REGION Network 6: #"PHT Selected"
   RUNG wire#powerrail
      Contact( #DataLogYes )
      I_Contact( #ScadaHmi )
      wire#w1
      I_Contact( #Popup2Enable )
      wire#w2
      I_Contact( #Stop )
      I_Contact( #Fault )
      I_Contact( #ReleaseCheckTime.DONE_BIT )
      wire#w3
      S_Coil( #"PHT Selected" )
   END_RUNG
   RUNG wire#powerrail
      Contact( #StartupMsgYes )
      Contact( #ScadaHmi )
   END_RUNG wire#w1
   RUNG wire#powerrail
      Contact( #Popup2Ack )
      Contact( #Popup2Enable )
   END_RUNG wire#w2
   RUNG wire#powerrail
      Contact( #"PHT Selected" )
      Contact( #Start )
   END_RUNG wire#w2
   RUNG wire#powerrail
      Contact( #Running )
   END_RUNG wire#w2
   RUNG wire#w3
      Coil( #Running )
   END_RUNG
   // the same network as SCL:
   #_w1 := ((((#DataLogYes AND NOT #ScadaHmi) OR (#StartupMsgYes AND #ScadaHmi)) AND NOT #Popup2Enable) OR (#Popup2Ack AND #Popup2Enable) OR (#"PHT Selected" AND #Start) OR #Running) AND NOT #Stop AND NOT #Fault AND NOT #ReleaseCheckTime.DONE_BIT;
   IF #_w1 THEN #"PHT Selected" := TRUE; END_IF;
   #Running := #_w1;
END_REGION

REGION Network 7
   RUNG wire#powerrail
      Contact( #AlwaysTrue )
      wire#w1
      Contact( #"PHT Selected" )
      wire#w2
      R_Coil( #StartLog )
   END_RUNG
   RUNG wire#w1
      I_Contact( #CycleSelected )
   END_RUNG wire#w2
   RUNG wire#w1
      I_Contact( #"PHT Selected" )
      R_Coil( #EndLog )
   END_RUNG
   // the same network as SCL:
   IF #AlwaysTrue AND (#"PHT Selected" OR NOT #CycleSelected) THEN #StartLog := FALSE; END_IF;
   IF #AlwaysTrue AND NOT #"PHT Selected" THEN #EndLog := FALSE; END_IF;
END_REGION

REGION Network 8: OUTPUT ON
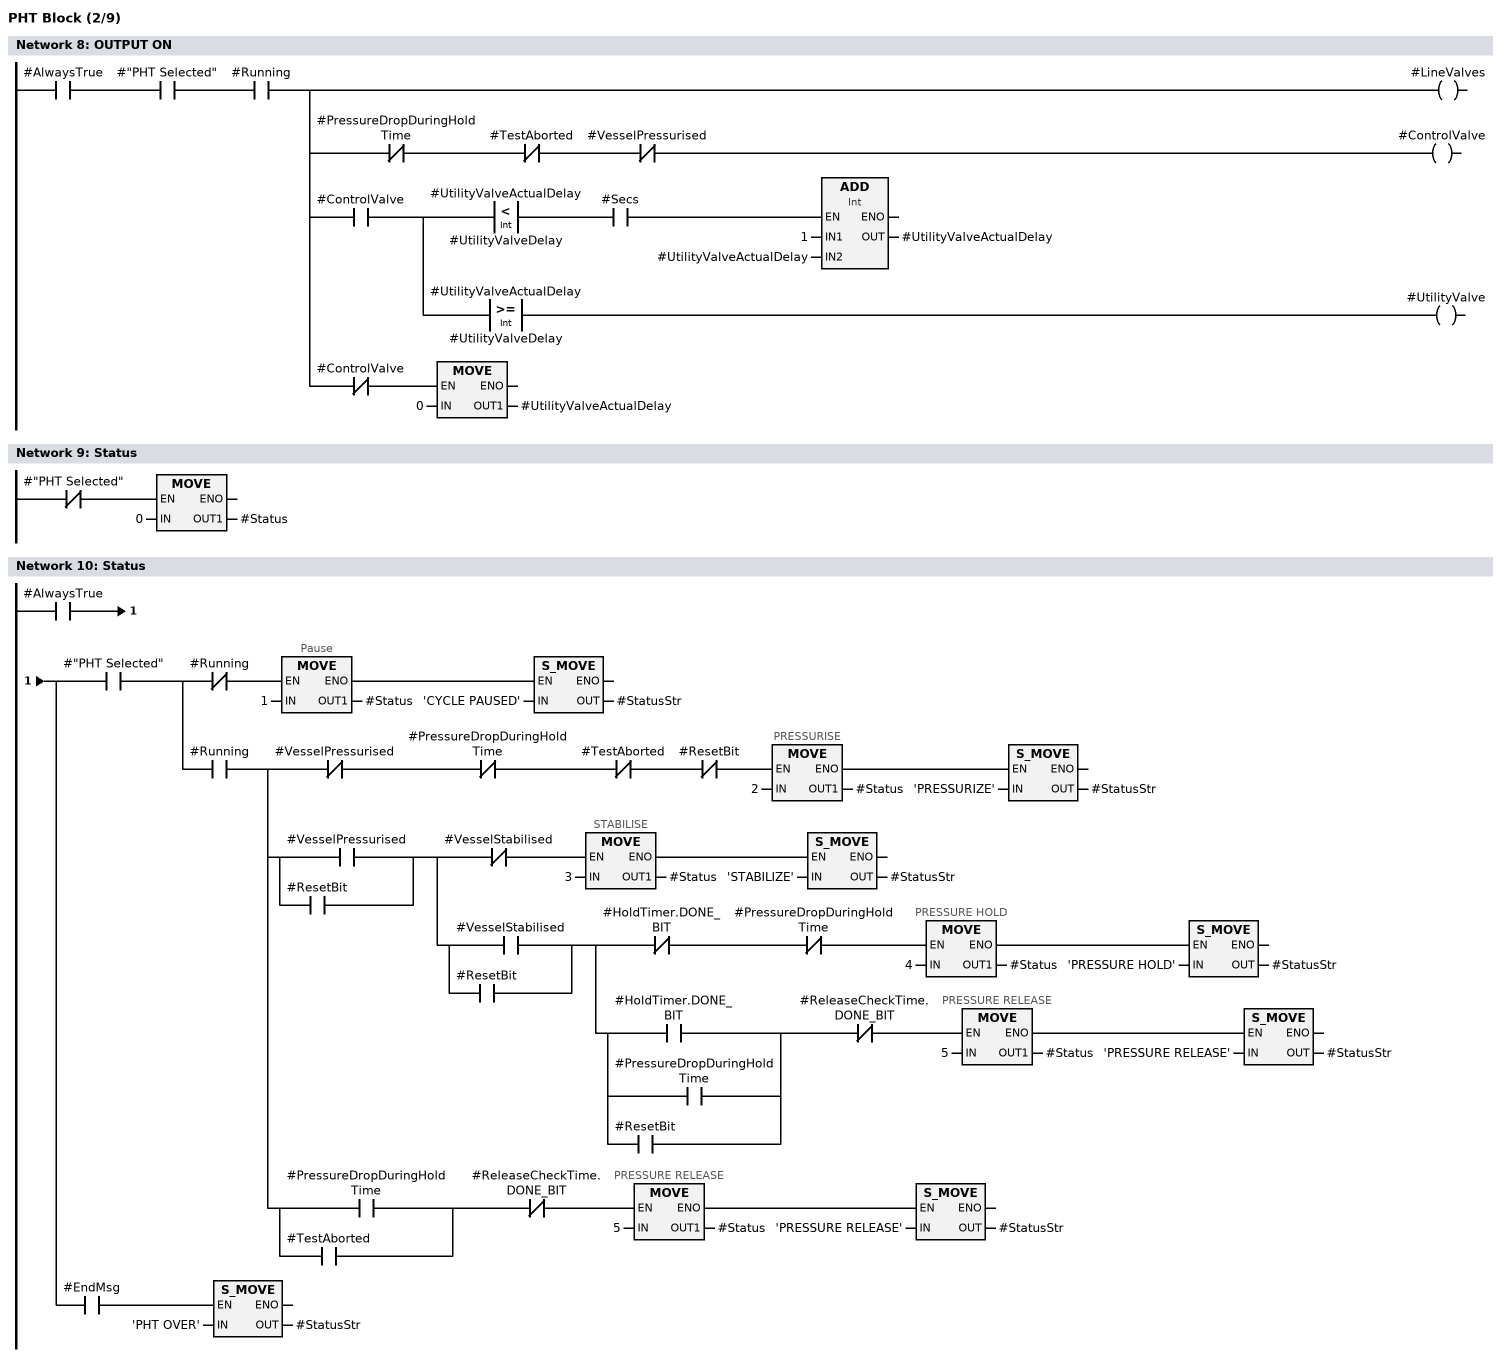
   RUNG wire#powerrail
      Contact( #AlwaysTrue )
      Contact( #"PHT Selected" )
      Contact( #Running )
      wire#w1
      Coil( #LineValves )
   END_RUNG
   RUNG wire#w1
      I_Contact( #PressureDropDuringHoldTime )
      I_Contact( #TestAborted )
      I_Contact( #VesselPressurised )
      Coil( #ControlValve )
   END_RUNG
   RUNG wire#w1
      Contact( #ControlValve )
      wire#w2
      { S7_Templates := "SrcType := Int" } LT_Contact(in1 := #UtilityValveActualDelay, in2 := #UtilityValveDelay)
      Contact( #Secs )
      { S7_Templates := "SrcType := Int" } Add(in1 := 1, in2 := #UtilityValveActualDelay, out => #UtilityValveActualDelay)
   END_RUNG
   RUNG wire#w2
      { S7_Templates := "SrcType := Int" } GE_Contact(in1 := #UtilityValveActualDelay, in2 := #UtilityValveDelay)
      Coil( #UtilityValve )
   END_RUNG
   RUNG wire#w1
      I_Contact( #ControlValve )
      Move(in := 0, out1 => #UtilityValveActualDelay)
   END_RUNG
   // the same network as SCL:
   #LineValves := #AlwaysTrue AND #"PHT Selected" AND #Running;
   #ControlValve := #LineValves AND NOT #PressureDropDuringHoldTime AND NOT #TestAborted AND NOT #VesselPressurised;
   #_w1 := #LineValves AND #ControlValve;
   IF #_w1 AND (#UtilityValveActualDelay < #UtilityValveDelay) AND #Secs THEN
       #UtilityValveActualDelay := 1 + #UtilityValveActualDelay;
   END_IF;
   #UtilityValve := #_w1 AND (#UtilityValveActualDelay >= #UtilityValveDelay);
   IF #LineValves AND NOT #ControlValve THEN #UtilityValveActualDelay := 0; END_IF;
END_REGION

REGION Network 9: Status
   RUNG wire#powerrail
      I_Contact( #"PHT Selected" )
      { S7_GenerateENO := "TRUE" } Move(in := 0, out1 => #Status)
   END_RUNG
   // the same network as SCL:
   IF NOT #"PHT Selected" THEN #Status := 0; END_IF;
END_REGION

REGION Network 10: Status
   RUNG wire#powerrail
      Contact( #AlwaysTrue )
      wire#w1
      Contact( #"PHT Selected" )
      wire#w2
      I_Contact( #Running )
      { S7_GenerateENO := "TRUE" } Move(in := 1, out1 => #Status)   // Pause
      S_Move(in := 'CYCLE PAUSED', out => #StatusStr)
   END_RUNG
   RUNG wire#w2
      Contact( #Running )
      wire#w3
      I_Contact( #VesselPressurised )
      I_Contact( #PressureDropDuringHoldTime )
      I_Contact( #TestAborted )
      I_Contact( #ResetBit )
      { S7_GenerateENO := "TRUE" } Move(in := 2, out1 => #Status)   // PRESSURISE
      S_Move(in := 'PRESSURIZE', out => #StatusStr)
   END_RUNG
   RUNG wire#w3
      Contact( #VesselPressurised )
      wire#w4
      I_Contact( #VesselStabilised )
      { S7_GenerateENO := "TRUE" } Move(in := 3, out1 => #Status)   // STABILISE
      S_Move(in := 'STABILIZE', out => #StatusStr)
   END_RUNG
   RUNG wire#w3
      Contact( #ResetBit )
   END_RUNG wire#w4
   RUNG wire#w4
      Contact( #VesselStabilised )
      wire#w5
      I_Contact( #HoldTimer.DONE_BIT )
      I_Contact( #PressureDropDuringHoldTime )
      { S7_GenerateENO := "TRUE" } Move(in := 4, out1 => #Status)   // PRESSURE HOLD
      S_Move(in := 'PRESSURE HOLD', out => #StatusStr)
   END_RUNG
   RUNG wire#w4
      Contact( #ResetBit )
   END_RUNG wire#w5
   RUNG wire#w5
      Contact( #HoldTimer.DONE_BIT )
      wire#w6
      I_Contact( #ReleaseCheckTime.DONE_BIT )
      { S7_GenerateENO := "TRUE" } Move(in := 5, out1 => #Status)   // PRESSURE RELEASE
      S_Move(in := 'PRESSURE RELEASE', out => #StatusStr)
   END_RUNG
   RUNG wire#w5
      Contact( #PressureDropDuringHoldTime )
   END_RUNG wire#w6
   RUNG wire#w5
      Contact( #ResetBit )
   END_RUNG wire#w6
   RUNG wire#w3
      Contact( #PressureDropDuringHoldTime )
      wire#w7
      I_Contact( #ReleaseCheckTime.DONE_BIT )
      { S7_GenerateENO := "TRUE" } Move(in := 5, out1 => #Status)   // PRESSURE RELEASE
      S_Move(in := 'PRESSURE RELEASE', out => #StatusStr)
   END_RUNG
   RUNG wire#w3
      Contact( #TestAborted )
   END_RUNG wire#w7
   RUNG wire#w1
      Contact( #EndMsg )
      S_Move(in := 'PHT OVER', out => #StatusStr)
   END_RUNG
   // the same network as SCL:
   // ENO of a box is taken as its EN; it also drops when the box reports an error
   #_w1 := #AlwaysTrue AND #"PHT Selected";
   IF #_w1 AND NOT #Running THEN
       #Status := 1;   // Pause
       #StatusStr := 'CYCLE PAUSED';
   END_IF;
   #_w2 := #_w1 AND #Running;
   IF #_w2 AND NOT #VesselPressurised AND NOT #PressureDropDuringHoldTime AND NOT #TestAborted AND NOT #ResetBit THEN
       #Status := 2;   // PRESSURISE
       #StatusStr := 'PRESSURIZE';
   END_IF;
   #_w3 := #_w2 AND (#VesselPressurised OR #ResetBit);
   IF #_w3 AND NOT #VesselStabilised THEN
       #Status := 3;   // STABILISE
       #StatusStr := 'STABILIZE';
   END_IF;
   #_w4 := #_w3 AND (#VesselStabilised OR #ResetBit);
   IF #_w4 AND NOT #HoldTimer.DONE_BIT AND NOT #PressureDropDuringHoldTime THEN
       #Status := 4;   // PRESSURE HOLD
       #StatusStr := 'PRESSURE HOLD';
   END_IF;
   IF #_w4 AND (#HoldTimer.DONE_BIT OR #PressureDropDuringHoldTime OR #ResetBit) AND NOT #ReleaseCheckTime.DONE_BIT THEN
       #Status := 5;   // PRESSURE RELEASE
       #StatusStr := 'PRESSURE RELEASE';
   END_IF;
   IF #_w2 AND (#PressureDropDuringHoldTime OR #TestAborted) AND NOT #ReleaseCheckTime.DONE_BIT THEN
       #Status := 5;   // PRESSURE RELEASE
       #StatusStr := 'PRESSURE RELEASE';
   END_IF;
   IF #AlwaysTrue AND #EndMsg THEN #StatusStr := 'PHT OVER'; END_IF;
END_REGION

REGION Network 11: Delays for opening drain valves
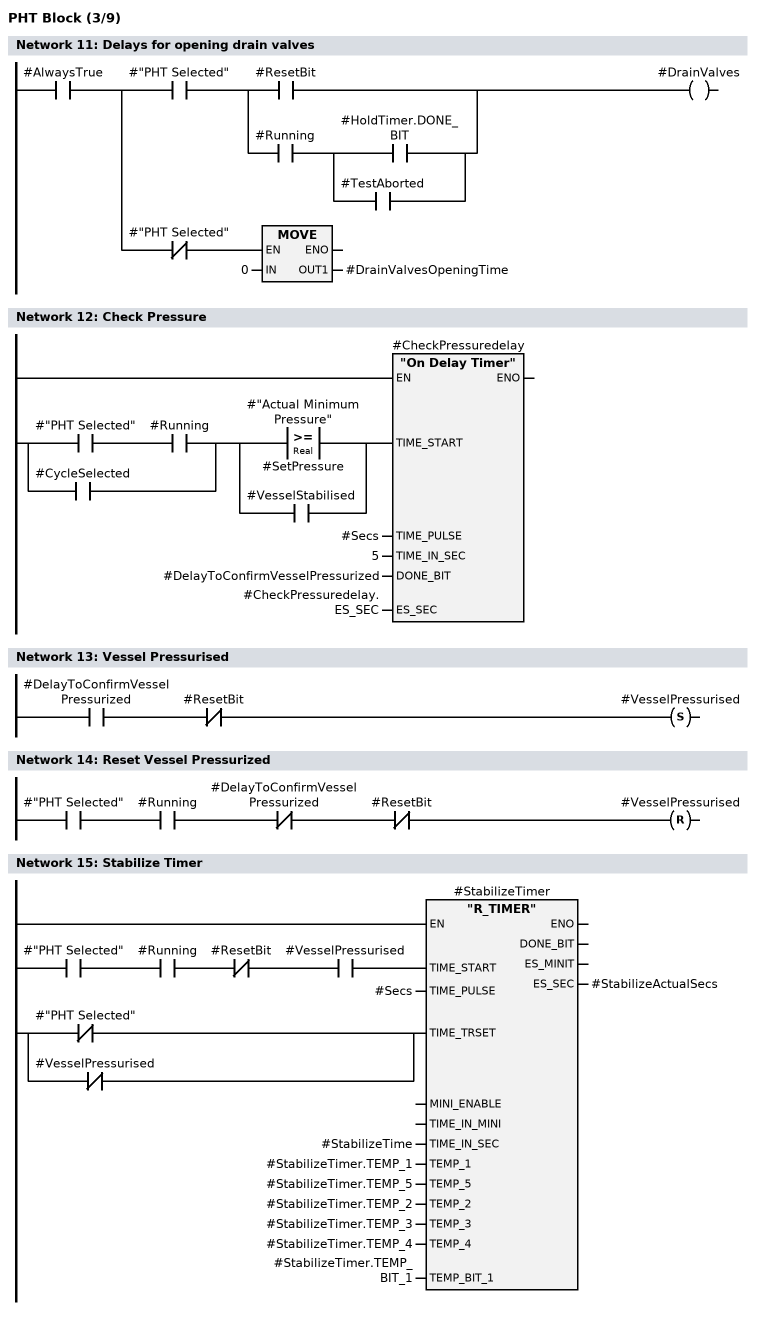
   RUNG wire#powerrail
      Contact( #AlwaysTrue )
      wire#w1
      Contact( #"PHT Selected" )
      wire#w2
      Contact( #ResetBit )
      wire#w3
      Coil( #DrainValves )
   END_RUNG
   RUNG wire#w2
      Contact( #Running )
      wire#w4
      Contact( #HoldTimer.DONE_BIT )
   END_RUNG wire#w3
   RUNG wire#w4
      Contact( #TestAborted )
   END_RUNG wire#w3
   RUNG wire#w1
      I_Contact( #"PHT Selected" )
      { S7_GenerateENO := "TRUE" } Move(in := 0, out1 => #DrainValvesOpeningTime)
   END_RUNG
   // the same network as SCL:
   #DrainValves := #AlwaysTrue AND #"PHT Selected" AND (#ResetBit OR (#Running AND (#HoldTimer.DONE_BIT OR #TestAborted)));
   IF #AlwaysTrue AND NOT #"PHT Selected" THEN #DrainValvesOpeningTime := 0; END_IF;
END_REGION

REGION Network 12: Check Pressure
   RUNG wire#powerrail
      #CheckPressuredelay(TIME_START := wire#w2, TIME_PULSE := #Secs, TIME_IN_SEC := 5, DONE_BIT := #DelayToConfirmVesselPressurized, ES_SEC := #CheckPressuredelay.ES_SEC)
   END_RUNG
   RUNG wire#powerrail
      Contact( #"PHT Selected" )
      Contact( #Running )
      wire#w1
      { S7_Templates := "SrcType := Real" } GE_Contact(in1 := #"Actual Minimum Pressure", in2 := #SetPressure)
   END_RUNG wire#w2
   RUNG wire#powerrail
      Contact( #CycleSelected )
   END_RUNG wire#w1
   RUNG wire#w1
      Contact( #VesselStabilised )
   END_RUNG wire#w2
   // the same network as SCL:
   #CheckPressuredelay(TIME_START := ((#"PHT Selected" AND #Running) OR #CycleSelected) AND ((#"Actual Minimum Pressure" >= #SetPressure) OR #VesselStabilised),   // "On Delay Timer"
                       TIME_PULSE := #Secs,
                       TIME_IN_SEC := 5,
                       DONE_BIT := #DelayToConfirmVesselPressurized,
                       ES_SEC := #CheckPressuredelay.ES_SEC);
END_REGION

REGION Network 13: Vessel Pressurised
   RUNG wire#powerrail
      Contact( #DelayToConfirmVesselPressurized )
      I_Contact( #ResetBit )
      S_Coil( #VesselPressurised )
   END_RUNG
   // the same network as SCL:
   IF #DelayToConfirmVesselPressurized AND NOT #ResetBit THEN #VesselPressurised := TRUE; END_IF;
END_REGION

REGION Network 14: Reset Vessel Pressurized
   RUNG wire#powerrail
      Contact( #"PHT Selected" )
      Contact( #Running )
      I_Contact( #DelayToConfirmVesselPressurized )
      I_Contact( #ResetBit )
      R_Coil( #VesselPressurised )
   END_RUNG
   // the same network as SCL:
   IF #"PHT Selected" AND #Running AND NOT #DelayToConfirmVesselPressurized AND NOT #ResetBit THEN
       #VesselPressurised := FALSE;
   END_IF;
END_REGION

REGION Network 15: Stabilize Timer
   RUNG wire#powerrail
      #StabilizeTimer(TIME_START := wire#w1, TIME_TRSET := wire#w2, TIME_PULSE := #Secs, MINI_ENABLE :=, TIME_IN_MINI :=, TIME_IN_SEC := #StabilizeTime, TEMP_1 := #StabilizeTimer.TEMP_1, TEMP_5 := #StabilizeTimer.TEMP_5, TEMP_2 := #StabilizeTimer.TEMP_2, TEMP_3 := #StabilizeTimer.TEMP_3, TEMP_4 := #StabilizeTimer.TEMP_4, TEMP_BIT_1 := #StabilizeTimer.TEMP_BIT_1, DONE_BIT =>, ES_MINIT =>, ES_SEC => #StabilizeActualSecs)
   END_RUNG
   RUNG wire#powerrail
      Contact( #"PHT Selected" )
      Contact( #Running )
      I_Contact( #ResetBit )
      Contact( #VesselPressurised )
   END_RUNG wire#w1
   RUNG wire#powerrail
      I_Contact( #"PHT Selected" )
   END_RUNG wire#w2
   RUNG wire#powerrail
      I_Contact( #VesselPressurised )
   END_RUNG wire#w2
   // the same network as SCL:
   #StabilizeTimer(TIME_START := #"PHT Selected" AND #Running AND NOT #ResetBit AND #VesselPressurised,   // "R_TIMER"
                   TIME_PULSE := #Secs,
                   TIME_TRSET := NOT #"PHT Selected" OR NOT #VesselPressurised,
                   TIME_IN_SEC := #StabilizeTime,
                   TEMP_1 := #StabilizeTimer.TEMP_1,
                   TEMP_5 := #StabilizeTimer.TEMP_5,
                   TEMP_2 := #StabilizeTimer.TEMP_2,
                   TEMP_3 := #StabilizeTimer.TEMP_3,
                   TEMP_4 := #StabilizeTimer.TEMP_4,
                   TEMP_BIT_1 := #StabilizeTimer.TEMP_BIT_1,
                   ES_SEC => #StabilizeActualSecs);
END_REGION

REGION Network 16: Check Pressure During Stabilize
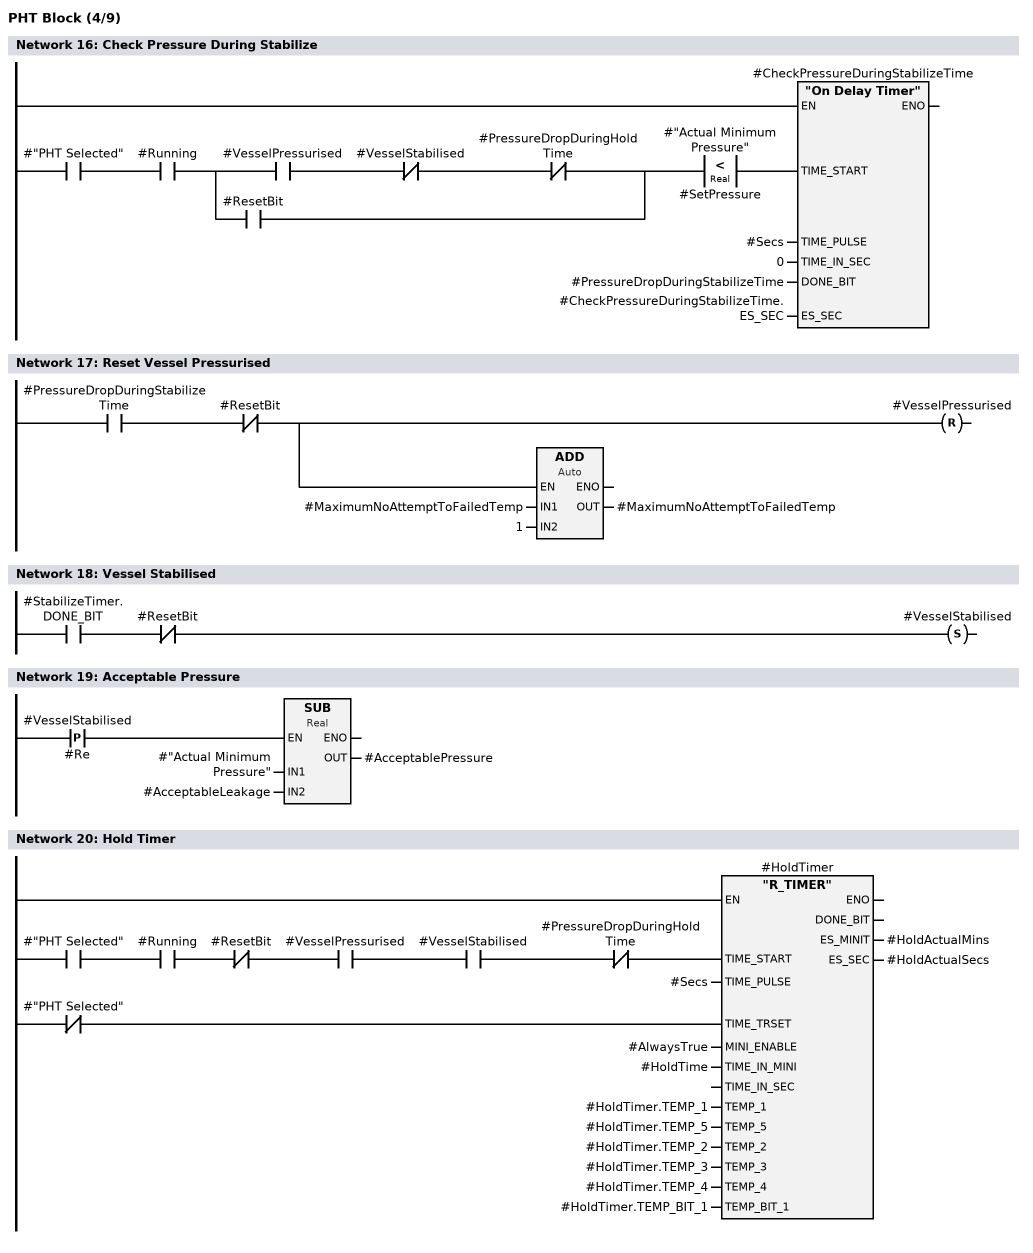
   RUNG wire#powerrail
      #CheckPressureDuringStabilizeTime(TIME_START := wire#w3, TIME_PULSE := #Secs, TIME_IN_SEC := 0, DONE_BIT := #PressureDropDuringStabilizeTime, ES_SEC := #CheckPressureDuringStabilizeTime.ES_SEC)
   END_RUNG
   RUNG wire#powerrail
      Contact( #"PHT Selected" )
      Contact( #Running )
      wire#w1
      Contact( #VesselPressurised )
      I_Contact( #VesselStabilised )
      I_Contact( #PressureDropDuringHoldTime )
      wire#w2
      { S7_Templates := "SrcType := Real" } LT_Contact(in1 := #"Actual Minimum Pressure", in2 := #SetPressure)
   END_RUNG wire#w3
   RUNG wire#w1
      Contact( #ResetBit )
   END_RUNG wire#w2
   // the same network as SCL:
   #CheckPressureDuringStabilizeTime(TIME_START := #"PHT Selected" AND #Running AND ((#VesselPressurised AND NOT #VesselStabilised AND NOT #PressureDropDuringHoldTime) OR #ResetBit) AND (#"Actual Minimum Pressure" < #SetPressure),   // "On Delay Timer"
                           TIME_PULSE := #Secs,
                           TIME_IN_SEC := 0,
                           DONE_BIT := #PressureDropDuringStabilizeTime,
                           ES_SEC := #CheckPressureDuringStabilizeTime.ES_SEC);
END_REGION

REGION Network 17: Reset Vessel Pressurised
   RUNG wire#powerrail
      Contact( #PressureDropDuringStabilizeTime )
      I_Contact( #ResetBit )
      wire#w1
      R_Coil( #VesselPressurised )
   END_RUNG
   RUNG wire#w1
      Add(in1 := #MaximumNoAttemptToFailedTemp, in2 := 1, out => #MaximumNoAttemptToFailedTemp)
   END_RUNG
   // the same network as SCL:
   IF #PressureDropDuringStabilizeTime AND NOT #ResetBit THEN
       #VesselPressurised := FALSE;
       #MaximumNoAttemptToFailedTemp := #MaximumNoAttemptToFailedTemp + 1;
   END_IF;
END_REGION

REGION Network 18: Vessel Stabilised
   RUNG wire#powerrail
      Contact( #StabilizeTimer.DONE_BIT )
      I_Contact( #ResetBit )
      S_Coil( #VesselStabilised )
   END_RUNG
   // the same network as SCL:
   IF #StabilizeTimer.DONE_BIT AND NOT #ResetBit THEN #VesselStabilised := TRUE; END_IF;
END_REGION

REGION Network 19: Acceptable Pressure
   RUNG wire#powerrail
      P_Contact(operand := #VesselStabilised, bit := #Re)
      { S7_Templates := "SrcType := Real"; S7_GenerateENO := "TRUE" } Sub(in1 := #"Actual Minimum Pressure", in2 := #AcceptableLeakage, out => #AcceptablePressure)
   END_RUNG
   // the same network as SCL:
   #_w1 := #VesselStabilised AND NOT #Re;   // rising edge of #VesselStabilised
   #Re := #VesselStabilised;
   IF #_w1 THEN #AcceptablePressure := #"Actual Minimum Pressure" - #AcceptableLeakage; END_IF;
END_REGION

REGION Network 20: Hold Timer
   RUNG wire#powerrail
      #HoldTimer(TIME_START := wire#w1, TIME_TRSET := wire#w2, TIME_PULSE := #Secs, MINI_ENABLE := #AlwaysTrue, TIME_IN_MINI := #HoldTime, TIME_IN_SEC :=, TEMP_1 := #HoldTimer.TEMP_1, TEMP_5 := #HoldTimer.TEMP_5, TEMP_2 := #HoldTimer.TEMP_2, TEMP_3 := #HoldTimer.TEMP_3, TEMP_4 := #HoldTimer.TEMP_4, TEMP_BIT_1 := #HoldTimer.TEMP_BIT_1, DONE_BIT =>, ES_MINIT => #HoldActualMins, ES_SEC => #HoldActualSecs)
   END_RUNG
   RUNG wire#powerrail
      Contact( #"PHT Selected" )
      Contact( #Running )
      I_Contact( #ResetBit )
      Contact( #VesselPressurised )
      Contact( #VesselStabilised )
      I_Contact( #PressureDropDuringHoldTime )
   END_RUNG wire#w1
   RUNG wire#powerrail
      I_Contact( #"PHT Selected" )
   END_RUNG wire#w2
   // the same network as SCL:
   #HoldTimer(TIME_START := #"PHT Selected" AND #Running AND NOT #ResetBit AND #VesselPressurised AND #VesselStabilised AND NOT #PressureDropDuringHoldTime,   // "R_TIMER"
              TIME_PULSE := #Secs,
              TIME_TRSET := NOT #"PHT Selected",
              MINI_ENABLE := #AlwaysTrue,
              TIME_IN_MINI := #HoldTime,
              TEMP_1 := #HoldTimer.TEMP_1,
              TEMP_5 := #HoldTimer.TEMP_5,
              TEMP_2 := #HoldTimer.TEMP_2,
              TEMP_3 := #HoldTimer.TEMP_3,
              TEMP_4 := #HoldTimer.TEMP_4,
              TEMP_BIT_1 := #HoldTimer.TEMP_BIT_1,
              ES_MINIT => #HoldActualMins,
              ES_SEC => #HoldActualSecs);
END_REGION

REGION Network 21: Check Pressure to abort Cycle during Hold Time
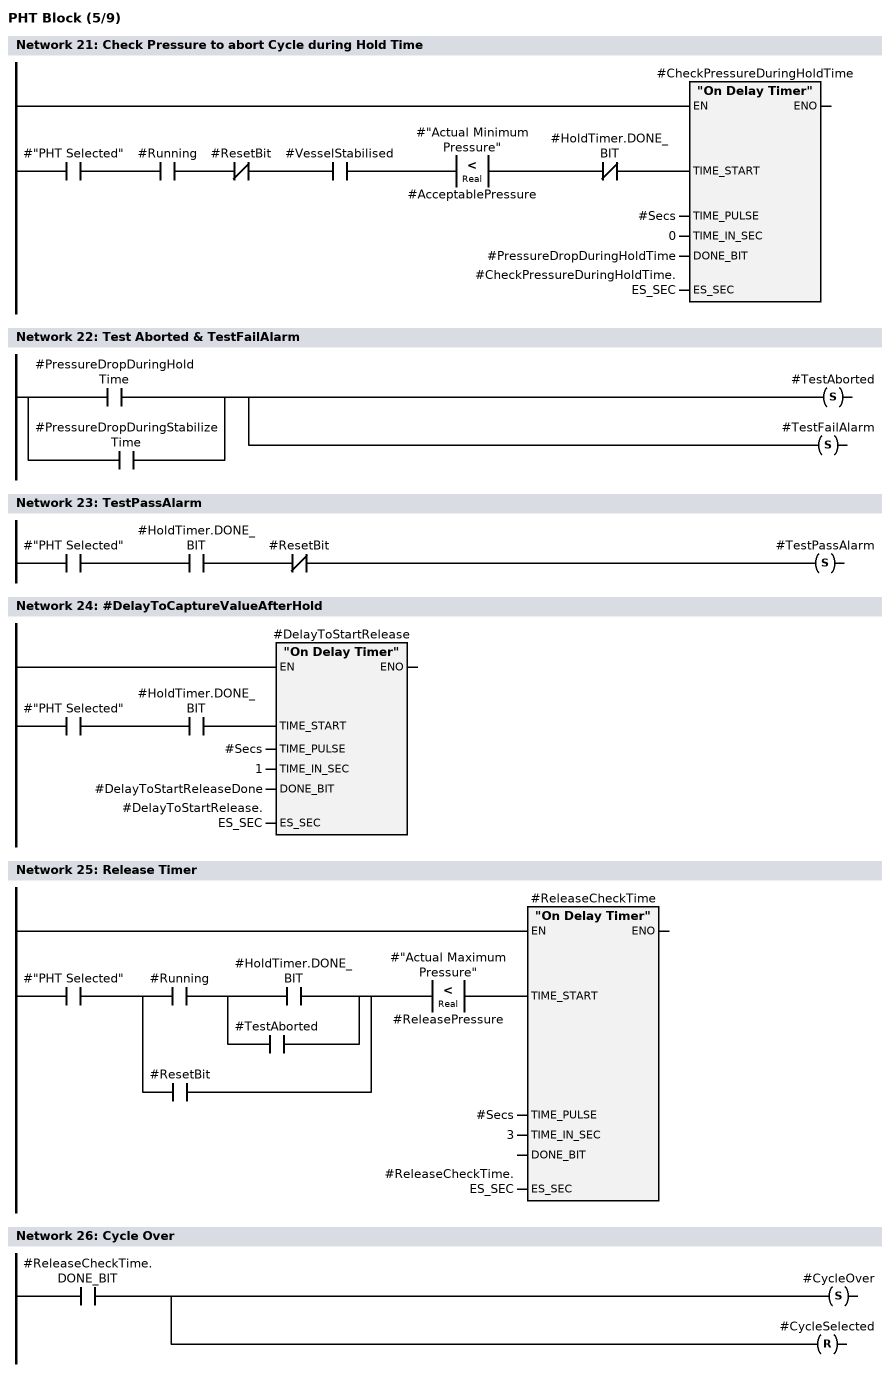
   RUNG wire#powerrail
      #CheckPressureDuringHoldTime(TIME_START := wire#w1, TIME_PULSE := #Secs, TIME_IN_SEC := 0, DONE_BIT := #PressureDropDuringHoldTime, ES_SEC := #CheckPressureDuringHoldTime.ES_SEC)
   END_RUNG
   RUNG wire#powerrail
      Contact( #"PHT Selected" )
      Contact( #Running )
      I_Contact( #ResetBit )
      Contact( #VesselStabilised )
      { S7_Templates := "SrcType := Real" } LT_Contact(in1 := #"Actual Minimum Pressure", in2 := #AcceptablePressure)
      I_Contact( #HoldTimer.DONE_BIT )
   END_RUNG wire#w1
   // the same network as SCL:
   #CheckPressureDuringHoldTime(TIME_START := #"PHT Selected" AND #Running AND NOT #ResetBit AND #VesselStabilised AND (#"Actual Minimum Pressure" < #AcceptablePressure) AND NOT #HoldTimer.DONE_BIT,   // "On Delay Timer"
                           TIME_PULSE := #Secs,
                           TIME_IN_SEC := 0,
                           DONE_BIT := #PressureDropDuringHoldTime,
                           ES_SEC := #CheckPressureDuringHoldTime.ES_SEC);
END_REGION

REGION Network 22: Test Aborted & TestFailAlarm
   RUNG wire#powerrail
      Contact( #PressureDropDuringHoldTime )
      wire#w1
      S_Coil( #TestAborted )
   END_RUNG
   RUNG wire#powerrail
      Contact( #PressureDropDuringStabilizeTime )
   END_RUNG wire#w1
   RUNG wire#w1
      S_Coil( #TestFailAlarm )
   END_RUNG
   // the same network as SCL:
   IF #PressureDropDuringHoldTime OR #PressureDropDuringStabilizeTime THEN
       #TestAborted := TRUE;
       #TestFailAlarm := TRUE;
   END_IF;
END_REGION

REGION Network 23: TestPassAlarm
   RUNG wire#powerrail
      Contact( #"PHT Selected" )
      Contact( #HoldTimer.DONE_BIT )
      I_Contact( #ResetBit )
      S_Coil( #TestPassAlarm )
   END_RUNG
   // the same network as SCL:
   IF #"PHT Selected" AND #HoldTimer.DONE_BIT AND NOT #ResetBit THEN #TestPassAlarm := TRUE; END_IF;
END_REGION

REGION Network 24: #DelayToCaptureValueAfterHold
   RUNG wire#powerrail
      #DelayToStartRelease(TIME_START := wire#w1, TIME_PULSE := #Secs, TIME_IN_SEC := 1, DONE_BIT := #DelayToStartReleaseDone, ES_SEC := #DelayToStartRelease.ES_SEC)
   END_RUNG
   RUNG wire#powerrail
      Contact( #"PHT Selected" )
      Contact( #HoldTimer.DONE_BIT )
   END_RUNG wire#w1
   // the same network as SCL:
   #DelayToStartRelease(TIME_START := #"PHT Selected" AND #HoldTimer.DONE_BIT,   // "On Delay Timer"
                        TIME_PULSE := #Secs,
                        TIME_IN_SEC := 1,
                        DONE_BIT := #DelayToStartReleaseDone,
                        ES_SEC := #DelayToStartRelease.ES_SEC);
END_REGION

REGION Network 25: Release Timer
   RUNG wire#powerrail
      #ReleaseCheckTime(TIME_START := wire#w4, TIME_PULSE := #Secs, TIME_IN_SEC := 3, DONE_BIT :=, ES_SEC := #ReleaseCheckTime.ES_SEC)
   END_RUNG
   RUNG wire#powerrail
      Contact( #"PHT Selected" )
      wire#w1
      Contact( #Running )
      wire#w2
      Contact( #HoldTimer.DONE_BIT )
      wire#w3
      { S7_Templates := "SrcType := Real" } LT_Contact(in1 := #"Actual Maximum Pressure", in2 := #ReleasePressure)
   END_RUNG wire#w4
   RUNG wire#w2
      Contact( #TestAborted )
   END_RUNG wire#w3
   RUNG wire#w1
      Contact( #ResetBit )
   END_RUNG wire#w3
   // the same network as SCL:
   #ReleaseCheckTime(TIME_START := #"PHT Selected" AND ((#Running AND (#HoldTimer.DONE_BIT OR #TestAborted)) OR #ResetBit) AND (#"Actual Maximum Pressure" < #ReleasePressure),   // "On Delay Timer"
                     TIME_PULSE := #Secs,
                     TIME_IN_SEC := 3,
                     ES_SEC := #ReleaseCheckTime.ES_SEC);
END_REGION

REGION Network 26: Cycle Over
   RUNG wire#powerrail
      Contact( #ReleaseCheckTime.DONE_BIT )
      wire#w1
      S_Coil( #CycleOver )
   END_RUNG
   RUNG wire#w1
      R_Coil( #CycleSelected )
   END_RUNG
   // the same network as SCL:
   IF #ReleaseCheckTime.DONE_BIT THEN
       #CycleOver := TRUE;
       #CycleSelected := FALSE;
   END_IF;
END_REGION

REGION Network 27: Alarm Ack
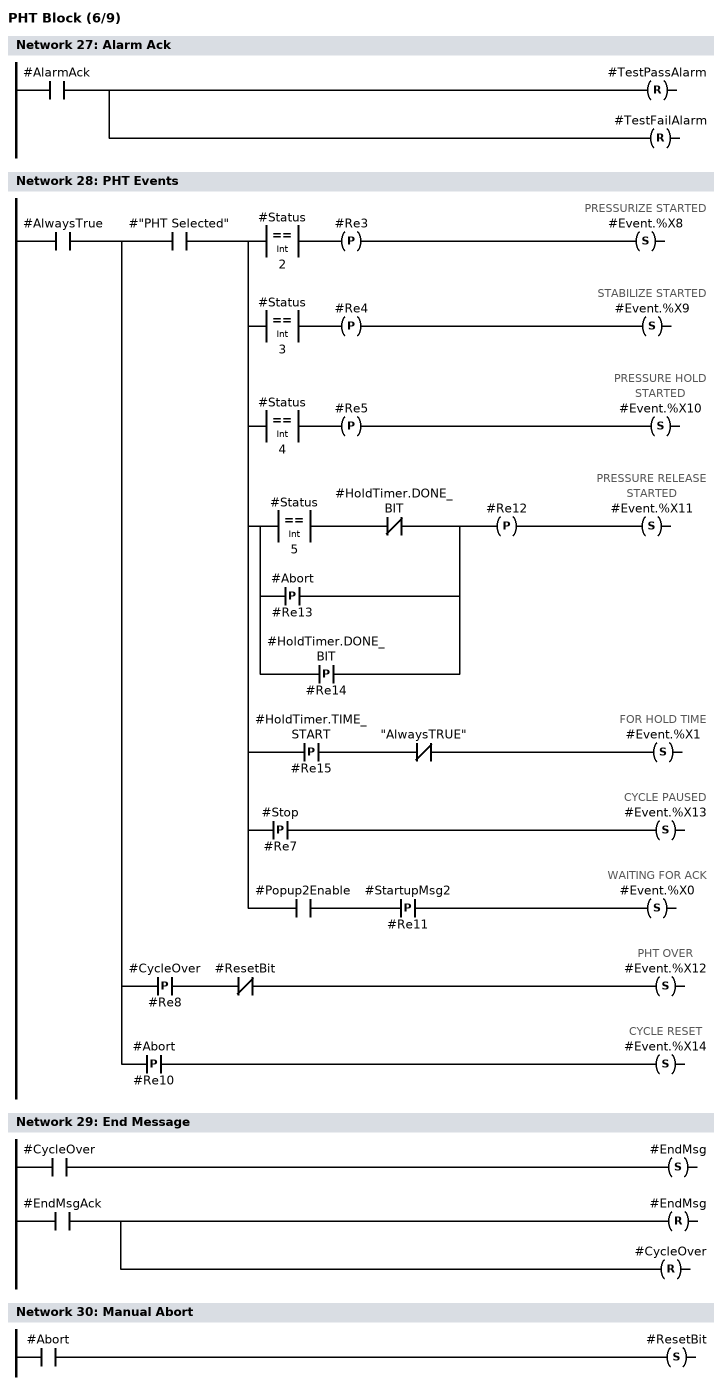
   RUNG wire#powerrail
      Contact( #AlarmAck )
      wire#w1
      R_Coil( #TestPassAlarm )
   END_RUNG
   RUNG wire#w1
      R_Coil( #TestFailAlarm )
   END_RUNG
   // the same network as SCL:
   IF #AlarmAck THEN
       #TestPassAlarm := FALSE;
       #TestFailAlarm := FALSE;
   END_IF;
END_REGION

REGION Network 28: PHT Events
   RUNG wire#powerrail
      Contact( #AlwaysTrue )
      wire#w1
      Contact( #"PHT Selected" )
      wire#w2
      { S7_Templates := "SrcType := Int" } EQ_Contact(in1 := #Status, in2 := 2)
      P_Trig( #Re3 )
      S_Coil( #Event.%X8 )   // PRESSURIZE STARTED
   END_RUNG
   RUNG wire#w2
      { S7_Templates := "SrcType := Int" } EQ_Contact(in1 := #Status, in2 := 3)
      P_Trig( #Re4 )
      S_Coil( #Event.%X9 )   // STABILIZE STARTED
   END_RUNG
   RUNG wire#w2
      { S7_Templates := "SrcType := Int" } EQ_Contact(in1 := #Status, in2 := 4)
      P_Trig( #Re5 )
      S_Coil( #Event.%X10 )   // PRESSURE HOLD STARTED
   END_RUNG
   RUNG wire#w2
      { S7_Templates := "SrcType := Int" } EQ_Contact(in1 := #Status, in2 := 5)
      I_Contact( #HoldTimer.DONE_BIT )
      wire#w3
      P_Trig( #Re12 )
      S_Coil( #Event.%X11 )   // PRESSURE RELEASE STARTED
   END_RUNG
   RUNG wire#w2
      P_Contact(operand := #Abort, bit := #Re13)
   END_RUNG wire#w3
   RUNG wire#w2
      P_Contact(operand := #HoldTimer.DONE_BIT, bit := #Re14)
   END_RUNG wire#w3
   RUNG wire#w2
      P_Contact(operand := #HoldTimer.TIME_START, bit := #Re15)
      I_Contact( "AlwaysTRUE" )
      S_Coil( #Event.%X1 )   // FOR HOLD TIME
   END_RUNG
   RUNG wire#w2
      P_Contact(operand := #Stop, bit := #Re7)
      S_Coil( #Event.%X13 )   // CYCLE PAUSED
   END_RUNG
   RUNG wire#w2
      Contact( #Popup2Enable )
      P_Contact(operand := #StartupMsg2, bit := #Re11)
      S_Coil( #Event.%X0 )   // WAITING FOR ACK
   END_RUNG
   RUNG wire#w1
      P_Contact(operand := #CycleOver, bit := #Re8)
      I_Contact( #ResetBit )
      S_Coil( #Event.%X12 )   // PHT OVER
   END_RUNG
   RUNG wire#w1
      P_Contact(operand := #Abort, bit := #Re10)
      S_Coil( #Event.%X14 )   // CYCLE RESET
   END_RUNG
   // the same network as SCL:
   #_w1 := #AlwaysTrue AND #"PHT Selected";
   #_w2 := #_w1 AND (#Status = 2);
   #_w3 := #_w2 AND NOT #Re3;   // rising edge
   #Re3 := #_w2;
   IF #_w3 THEN
       #Event.%X8 := TRUE;   // PRESSURIZE STARTED
   END_IF;
   #_w4 := #_w1 AND (#Status = 3);
   #_w5 := #_w4 AND NOT #Re4;   // rising edge
   #Re4 := #_w4;
   IF #_w5 THEN
       #Event.%X9 := TRUE;   // STABILIZE STARTED
   END_IF;
   #_w6 := #_w1 AND (#Status = 4);
   #_w7 := #_w6 AND NOT #Re5;   // rising edge
   #Re5 := #_w6;
   IF #_w7 THEN
       #Event.%X10 := TRUE;   // PRESSURE HOLD STARTED
   END_IF;
   #_w8 := #_w1 AND #Abort AND NOT #Re13;   // rising edge of #Abort
   #Re13 := #Abort;
   #_w9 := #_w1 AND #HoldTimer.DONE_BIT AND NOT #Re14;   // rising edge of #HoldTimer.DONE_BIT
   #Re14 := #HoldTimer.DONE_BIT;
   #_w10 := (#_w1 AND (#Status = 5) AND NOT #HoldTimer.DONE_BIT) OR #_w8 OR #_w9;
   #_w11 := #_w10 AND NOT #Re12;   // rising edge
   #Re12 := #_w10;
   IF #_w11 THEN
       #Event.%X11 := TRUE;   // PRESSURE RELEASE STARTED
   END_IF;
   #_w12 := #_w1 AND #HoldTimer.TIME_START AND NOT #Re15;   // rising edge of #HoldTimer.TIME_START
   #Re15 := #HoldTimer.TIME_START;
   IF #_w12 AND NOT "AlwaysTRUE" THEN
       #Event.%X1 := TRUE;   // FOR HOLD TIME
   END_IF;
   #_w13 := #_w1 AND #Stop AND NOT #Re7;   // rising edge of #Stop
   #Re7 := #Stop;
   IF #_w13 THEN
       #Event.%X13 := TRUE;   // CYCLE PAUSED
   END_IF;
   #_w14 := #_w1 AND #Popup2Enable AND #StartupMsg2 AND NOT #Re11;   // rising edge of #StartupMsg2
   #Re11 := #StartupMsg2;
   IF #_w14 THEN
       #Event.%X0 := TRUE;   // WAITING FOR ACK
   END_IF;
   #_w15 := #AlwaysTrue AND #CycleOver AND NOT #Re8;   // rising edge of #CycleOver
   #Re8 := #CycleOver;
   IF #_w15 AND NOT #ResetBit THEN
       #Event.%X12 := TRUE;   // PHT OVER
   END_IF;
   #_w16 := #AlwaysTrue AND #Abort AND NOT #Re10;   // rising edge of #Abort
   #Re10 := #Abort;
   IF #_w16 THEN
       #Event.%X14 := TRUE;   // CYCLE RESET
   END_IF;
END_REGION

REGION Network 29: End Message
   RUNG wire#powerrail
      Contact( #CycleOver )
      S_Coil( #EndMsg )
   END_RUNG
   RUNG wire#powerrail
      Contact( #EndMsgAck )
      wire#w1
      R_Coil( #EndMsg )
   END_RUNG
   RUNG wire#w1
      R_Coil( #CycleOver )
   END_RUNG
   // the same network as SCL:
   IF #CycleOver THEN #EndMsg := TRUE; END_IF;
   IF #EndMsgAck THEN
       #EndMsg := FALSE;
       #CycleOver := FALSE;
   END_IF;
END_REGION

REGION Network 30: Manual Abort
   RUNG wire#powerrail
      Contact( #Abort )
      S_Coil( #ResetBit )
   END_RUNG
   // the same network as SCL:
   IF #Abort THEN #ResetBit := TRUE; END_IF;
END_REGION

REGION Network 31: Reset
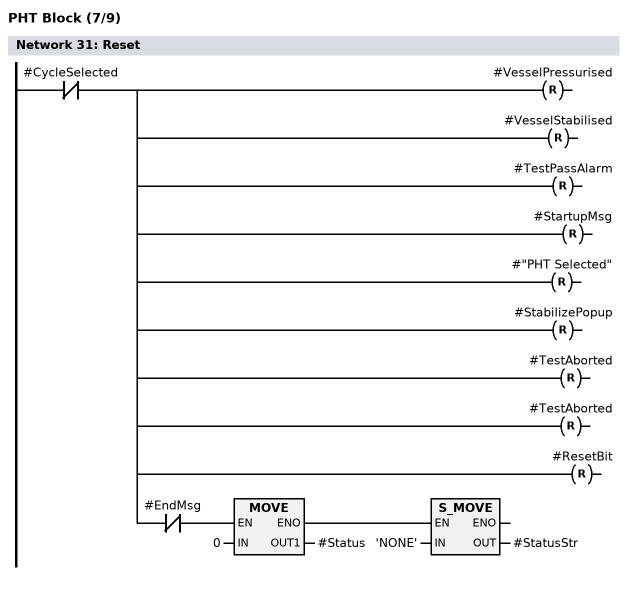
   RUNG wire#powerrail
      I_Contact( #CycleSelected )
      wire#w1
      R_Coil( #VesselPressurised )
   END_RUNG
   RUNG wire#w1
      R_Coil( #VesselStabilised )
   END_RUNG
   RUNG wire#w1
      R_Coil( #TestPassAlarm )
   END_RUNG
   RUNG wire#w1
      R_Coil( #StartupMsg )
   END_RUNG
   RUNG wire#w1
      R_Coil( #"PHT Selected" )
   END_RUNG
   RUNG wire#w1
      R_Coil( #StabilizePopup )
   END_RUNG
   RUNG wire#w1
      R_Coil( #TestAborted )
   END_RUNG
   RUNG wire#w1
      R_Coil( #TestAborted )
   END_RUNG
   RUNG wire#w1
      R_Coil( #ResetBit )
   END_RUNG
   RUNG wire#w1
      I_Contact( #EndMsg )
      { S7_GenerateENO := "TRUE" } Move(in := 0, out1 => #Status)
      S_Move(in := 'NONE', out => #StatusStr)
   END_RUNG
   // the same network as SCL:
   // ENO of a box is taken as its EN; it also drops when the box reports an error
   IF NOT #CycleSelected THEN
       #VesselPressurised := FALSE;
       #VesselStabilised := FALSE;
       #TestPassAlarm := FALSE;
       #StartupMsg := FALSE;
       #"PHT Selected" := FALSE;
       #StabilizePopup := FALSE;
       #TestAborted := FALSE;
       #TestAborted := FALSE;
       #ResetBit := FALSE;
   END_IF;
   IF NOT #CycleSelected AND NOT #EndMsg THEN
       #Status := 0;
       #StatusStr := 'NONE';
   END_IF;
END_REGION

REGION Network 32: Event reset
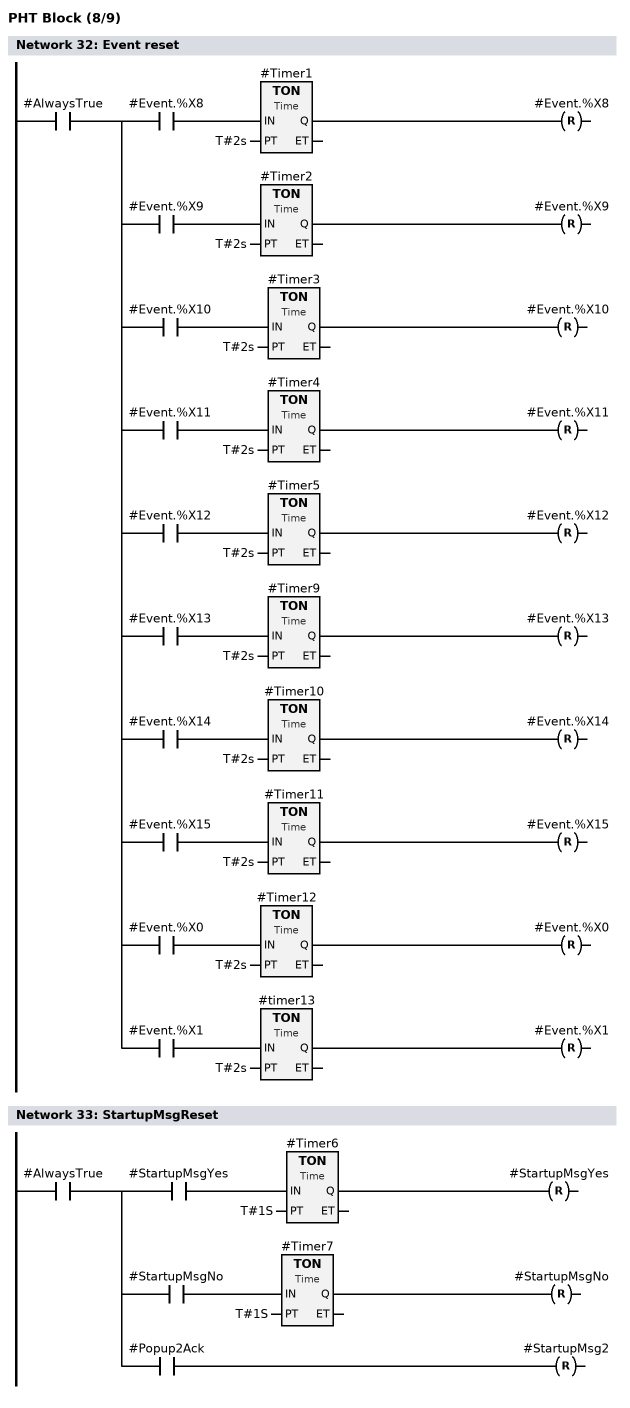
   RUNG wire#powerrail
      Contact( #AlwaysTrue )
      wire#w1
      Contact( #Event.%X8 )
      { S7_Templates := "time_type := Time" } #Timer1.TON(pt := T#2s, et =>)
      R_Coil( #Event.%X8 )
   END_RUNG
   RUNG wire#w1
      Contact( #Event.%X9 )
      { S7_Templates := "time_type := Time" } #Timer2.TON(pt := T#2s, et =>)
      R_Coil( #Event.%X9 )
   END_RUNG
   RUNG wire#w1
      Contact( #Event.%X10 )
      { S7_Templates := "time_type := Time" } #Timer3.TON(pt := T#2s, et =>)
      R_Coil( #Event.%X10 )
   END_RUNG
   RUNG wire#w1
      Contact( #Event.%X11 )
      { S7_Templates := "time_type := Time" } #Timer4.TON(pt := T#2s, et =>)
      R_Coil( #Event.%X11 )
   END_RUNG
   RUNG wire#w1
      Contact( #Event.%X12 )
      { S7_Templates := "time_type := Time" } #Timer5.TON(pt := T#2s, et =>)
      R_Coil( #Event.%X12 )
   END_RUNG
   RUNG wire#w1
      Contact( #Event.%X13 )
      { S7_Templates := "time_type := Time" } #Timer9.TON(pt := T#2s, et =>)
      R_Coil( #Event.%X13 )
   END_RUNG
   RUNG wire#w1
      Contact( #Event.%X14 )
      { S7_Templates := "time_type := Time" } #Timer10.TON(pt := T#2s, et =>)
      R_Coil( #Event.%X14 )
   END_RUNG
   RUNG wire#w1
      Contact( #Event.%X15 )
      { S7_Templates := "time_type := Time" } #Timer11.TON(pt := T#2s, et =>)
      R_Coil( #Event.%X15 )
   END_RUNG
   RUNG wire#w1
      Contact( #Event.%X0 )
      { S7_Templates := "time_type := Time" } #Timer12.TON(pt := T#2s, et =>)
      R_Coil( #Event.%X0 )
   END_RUNG
   RUNG wire#w1
      Contact( #Event.%X1 )
      { S7_Templates := "time_type := Time" } #timer13.TON(pt := T#2s, et =>)
      R_Coil( #Event.%X1 )
   END_RUNG
   // the same network as SCL:
   #Timer1(IN := #AlwaysTrue AND #Event.%X8, PT := T#2s);   // TON
   IF #Timer1.Q THEN #Event.%X8 := FALSE; END_IF;
   #Timer2(IN := #AlwaysTrue AND #Event.%X9, PT := T#2s);   // TON
   IF #Timer2.Q THEN #Event.%X9 := FALSE; END_IF;
   #Timer3(IN := #AlwaysTrue AND #Event.%X10, PT := T#2s);   // TON
   IF #Timer3.Q THEN #Event.%X10 := FALSE; END_IF;
   #Timer4(IN := #AlwaysTrue AND #Event.%X11, PT := T#2s);   // TON
   IF #Timer4.Q THEN #Event.%X11 := FALSE; END_IF;
   #Timer5(IN := #AlwaysTrue AND #Event.%X12, PT := T#2s);   // TON
   IF #Timer5.Q THEN #Event.%X12 := FALSE; END_IF;
   #Timer9(IN := #AlwaysTrue AND #Event.%X13, PT := T#2s);   // TON
   IF #Timer9.Q THEN #Event.%X13 := FALSE; END_IF;
   #Timer10(IN := #AlwaysTrue AND #Event.%X14, PT := T#2s);   // TON
   IF #Timer10.Q THEN #Event.%X14 := FALSE; END_IF;
   #Timer11(IN := #AlwaysTrue AND #Event.%X15, PT := T#2s);   // TON
   IF #Timer11.Q THEN #Event.%X15 := FALSE; END_IF;
   #Timer12(IN := #AlwaysTrue AND #Event.%X0, PT := T#2s);   // TON
   IF #Timer12.Q THEN #Event.%X0 := FALSE; END_IF;
   #timer13(IN := #AlwaysTrue AND #Event.%X1, PT := T#2s);   // TON
   IF #timer13.Q THEN #Event.%X1 := FALSE; END_IF;
END_REGION

REGION Network 33: StartupMsgReset
   RUNG wire#powerrail
      Contact( #AlwaysTrue )
      wire#w1
      Contact( #StartupMsgYes )
      { S7_Templates := "time_type := Time" } #Timer6.TON(pt := T#1S, et =>)
      R_Coil( #StartupMsgYes )
   END_RUNG
   RUNG wire#w1
      Contact( #StartupMsgNo )
      { S7_Templates := "time_type := Time" } #Timer7.TON(pt := T#1S, et =>)
      R_Coil( #StartupMsgNo )
   END_RUNG
   RUNG wire#w1
      Contact( #Popup2Ack )
      R_Coil( #StartupMsg2 )
   END_RUNG
   // the same network as SCL:
   #Timer6(IN := #AlwaysTrue AND #StartupMsgYes, PT := T#1S);   // TON
   IF #Timer6.Q THEN #StartupMsgYes := FALSE; END_IF;
   #Timer7(IN := #AlwaysTrue AND #StartupMsgNo, PT := T#1S);   // TON
   IF #Timer7.Q THEN #StartupMsgNo := FALSE; END_IF;
   IF #AlwaysTrue AND #Popup2Ack THEN #StartupMsg2 := FALSE; END_IF;
END_REGION

REGION Network 35: Line Print interval
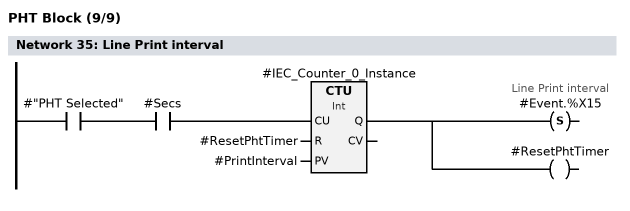
   RUNG wire#powerrail
      Contact( #"PHT Selected" )
      Contact( #Secs )
      { S7_Templates := "value_type := Int" } #IEC_Counter_0_Instance.CTU(r := #ResetPhtTimer, pv := #PrintInterval, cv =>)
      wire#w1
      S_Coil( #Event.%X15 )   // Line Print interval
   END_RUNG
   RUNG wire#w1
      Coil( #ResetPhtTimer )
   END_RUNG
   // the same network as SCL:
   #IEC_Counter_0_Instance(CU := #"PHT Selected" AND #Secs, R := #ResetPhtTimer, PV := #PrintInterval);   // CTU
   IF #IEC_Counter_0_Instance.Q THEN
       #Event.%X15 := TRUE;   // Line Print interval
   END_IF;
   #ResetPhtTimer := #IEC_Counter_0_Instance.Q;
END_REGION
END_FUNCTION_BLOCK

FUNCTION_BLOCK "On Delay Timer"   // FB150, LAD
{ S7_Optimized_Access := 'FALSE' }
// stored: AutoNumber false, SetENOAutomatically false
   VAR_INPUT
      TIME_START : Bool;
      TIME_PULSE : Bool;
      TIME_IN_SEC : Int;
   END_VAR
   VAR_IN_OUT
      DONE_BIT : Bool;
      ES_SEC : Int;
   END_VAR
   VAR_TEMP   // added for the SCL form of the ladder/FBD networks
      _w1 : Bool;
   END_VAR
BEGIN

REGION Network 1
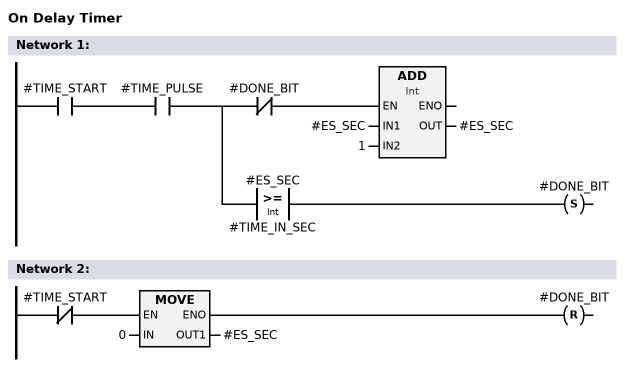
   RUNG wire#powerrail
      Contact( #TIME_START )
      Contact( #TIME_PULSE )
      wire#w1
      I_Contact( #DONE_BIT )
      { S7_Templates := "SrcType := Int"; S7_GenerateENO := "TRUE" } Add(in1 := #ES_SEC, in2 := 1, out => #ES_SEC)
   END_RUNG
   RUNG wire#w1
      { S7_Templates := "SrcType := Int" } GE_Contact(in1 := #ES_SEC, in2 := #TIME_IN_SEC)
      S_Coil( #DONE_BIT )
   END_RUNG
   // the same network as SCL:
   #_w1 := #TIME_START AND #TIME_PULSE;
   IF #_w1 AND NOT #DONE_BIT THEN #ES_SEC := #ES_SEC + 1; END_IF;
   IF #_w1 AND (#ES_SEC >= #TIME_IN_SEC) THEN #DONE_BIT := TRUE; END_IF;
END_REGION

REGION Network 2
   RUNG wire#powerrail
      I_Contact( #TIME_START )
      { S7_GenerateENO := "TRUE" } Move(in := 0, out1 => #ES_SEC)
      R_Coil( #DONE_BIT )
   END_RUNG
   // the same network as SCL:
   // ENO of a box is taken as its EN; it also drops when the box reports an error
   IF NOT #TIME_START THEN
       #ES_SEC := 0;
       #DONE_BIT := FALSE;
   END_IF;
END_REGION
END_FUNCTION_BLOCK

FUNCTION_BLOCK "R_TIMER"   // FB1, LAD
{ S7_Optimized_Access := 'FALSE' }
// stored: AutoNumber false, SetENOAutomatically false
   VAR_INPUT
      TIME_START : Bool;
      TIME_PULSE : Bool;
      TIME_TRSET : Bool;
      MINI_ENABLE : Bool;
      TIME_IN_MINI : Int;
      TIME_IN_SEC : Int;
   END_VAR
   VAR_OUTPUT
      DONE_BIT : Bool;
      ES_MINIT : DInt;
      ES_SEC : DInt;
   END_VAR
   VAR_IN_OUT
      TEMP_1 : Int;
      TEMP_5 : Int;
      TEMP_2 : Int;
      TEMP_3 : Int;
      TEMP_4 : DInt;
      TEMP_BIT_1 : Bool;
   END_VAR
BEGIN

REGION Network 1
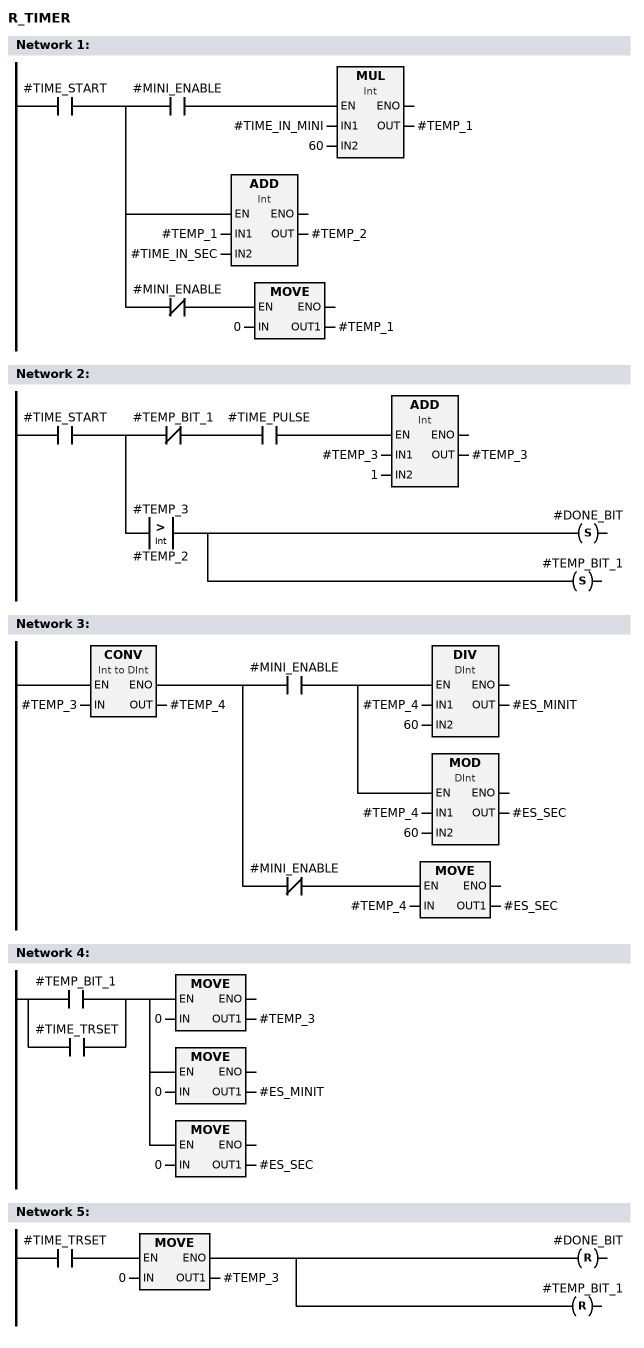
   RUNG wire#powerrail
      Contact( #TIME_START )
      wire#w1
      Contact( #MINI_ENABLE )
      { S7_Templates := "SrcType := Int"; S7_GenerateENO := "TRUE" } Mul(in1 := #TIME_IN_MINI, in2 := 60, out => #TEMP_1)
   END_RUNG
   RUNG wire#w1
      { S7_Templates := "SrcType := Int"; S7_GenerateENO := "TRUE" } Add(in1 := #TEMP_1, in2 := #TIME_IN_SEC, out => #TEMP_2)
   END_RUNG
   RUNG wire#w1
      I_Contact( #MINI_ENABLE )
      { S7_GenerateENO := "TRUE" } Move(in := 0, out1 => #TEMP_1)
   END_RUNG
   // the same network as SCL:
   IF #TIME_START AND #MINI_ENABLE THEN #TEMP_1 := #TIME_IN_MINI * 60; END_IF;
   IF #TIME_START THEN #TEMP_2 := #TEMP_1 + #TIME_IN_SEC; END_IF;
   IF #TIME_START AND NOT #MINI_ENABLE THEN #TEMP_1 := 0; END_IF;
END_REGION

REGION Network 2
   RUNG wire#powerrail
      Contact( #TIME_START )
      wire#w1
      I_Contact( #TEMP_BIT_1 )
      Contact( #TIME_PULSE )
      { S7_Templates := "SrcType := Int"; S7_GenerateENO := "TRUE" } Add(in1 := #TEMP_3, in2 := 1, out => #TEMP_3)
   END_RUNG
   RUNG wire#w1
      { S7_Templates := "SrcType := Int" } GT_Contact(in1 := #TEMP_3, in2 := #TEMP_2)
      wire#w2
      S_Coil( #DONE_BIT )
   END_RUNG
   RUNG wire#w2
      S_Coil( #TEMP_BIT_1 )
   END_RUNG
   // the same network as SCL:
   IF #TIME_START AND NOT #TEMP_BIT_1 AND #TIME_PULSE THEN #TEMP_3 := #TEMP_3 + 1; END_IF;
   IF #TIME_START AND (#TEMP_3 > #TEMP_2) THEN
       #DONE_BIT := TRUE;
       #TEMP_BIT_1 := TRUE;
   END_IF;
END_REGION

REGION Network 3
   RUNG wire#powerrail
      { S7_Templates := "[SrcType := Int, DestType := DInt]"; S7_GenerateENO := "TRUE" } Convert(in := #TEMP_3, out => #TEMP_4)
      wire#w1
      Contact( #MINI_ENABLE )
      wire#w2
      { S7_Templates := "SrcType := DInt"; S7_GenerateENO := "TRUE" } Div(in1 := #TEMP_4, in2 := 60, out => #ES_MINIT)
   END_RUNG
   RUNG wire#w2
      { S7_Templates := "SrcType := DInt"; S7_GenerateENO := "TRUE" } Mod(in1 := #TEMP_4, in2 := 60, out => #ES_SEC)
   END_RUNG
   RUNG wire#w1
      I_Contact( #MINI_ENABLE )
      { S7_GenerateENO := "TRUE" } Move(in := #TEMP_4, out1 => #ES_SEC)
   END_RUNG
   // the same network as SCL:
   // ENO of a box is taken as its EN; it also drops when the box reports an error
   #TEMP_4 := INT_TO_DINT(#TEMP_3);
   IF #MINI_ENABLE THEN
       #ES_MINIT := #TEMP_4 / 60;
       #ES_SEC := #TEMP_4 MOD 60;
   END_IF;
   IF NOT #MINI_ENABLE THEN #ES_SEC := #TEMP_4; END_IF;
END_REGION

REGION Network 4
   RUNG wire#powerrail
      Contact( #TEMP_BIT_1 )
      wire#w1
      { S7_GenerateENO := "TRUE" } Move(in := 0, out1 => #TEMP_3)
   END_RUNG
   RUNG wire#powerrail
      Contact( #TIME_TRSET )
   END_RUNG wire#w1
   RUNG wire#w1
      { S7_GenerateENO := "TRUE" } Move(in := 0, out1 => #ES_MINIT)
   END_RUNG
   RUNG wire#w1
      { S7_GenerateENO := "TRUE" } Move(in := 0, out1 => #ES_SEC)
   END_RUNG
   // the same network as SCL:
   IF #TEMP_BIT_1 OR #TIME_TRSET THEN
       #TEMP_3 := 0;
       #ES_MINIT := 0;
       #ES_SEC := 0;
   END_IF;
END_REGION

REGION Network 5
   RUNG wire#powerrail
      Contact( #TIME_TRSET )
      { S7_GenerateENO := "TRUE" } Move(in := 0, out1 => #TEMP_3)
      wire#w1
      R_Coil( #DONE_BIT )
   END_RUNG
   RUNG wire#w1
      R_Coil( #TEMP_BIT_1 )
   END_RUNG
   // the same network as SCL:
   // ENO of a box is taken as its EN; it also drops when the box reports an error
   IF #TIME_TRSET THEN
       #TEMP_3 := 0;
       #DONE_BIT := FALSE;
       #TEMP_BIT_1 := FALSE;
   END_IF;
END_REGION
END_FUNCTION_BLOCK

FUNCTION "PHT_ValveLogic" : Void   // FC1207, LAD
{ S7_Optimized_Access := 'TRUE' }
// stored: AutoNumber false, SetENOAutomatically false
BEGIN

REGION Network 1: ________________________________LINE VALVE________________________________
END_REGION

REGION Network 2: "PhtCycle".Cv24 - CAI
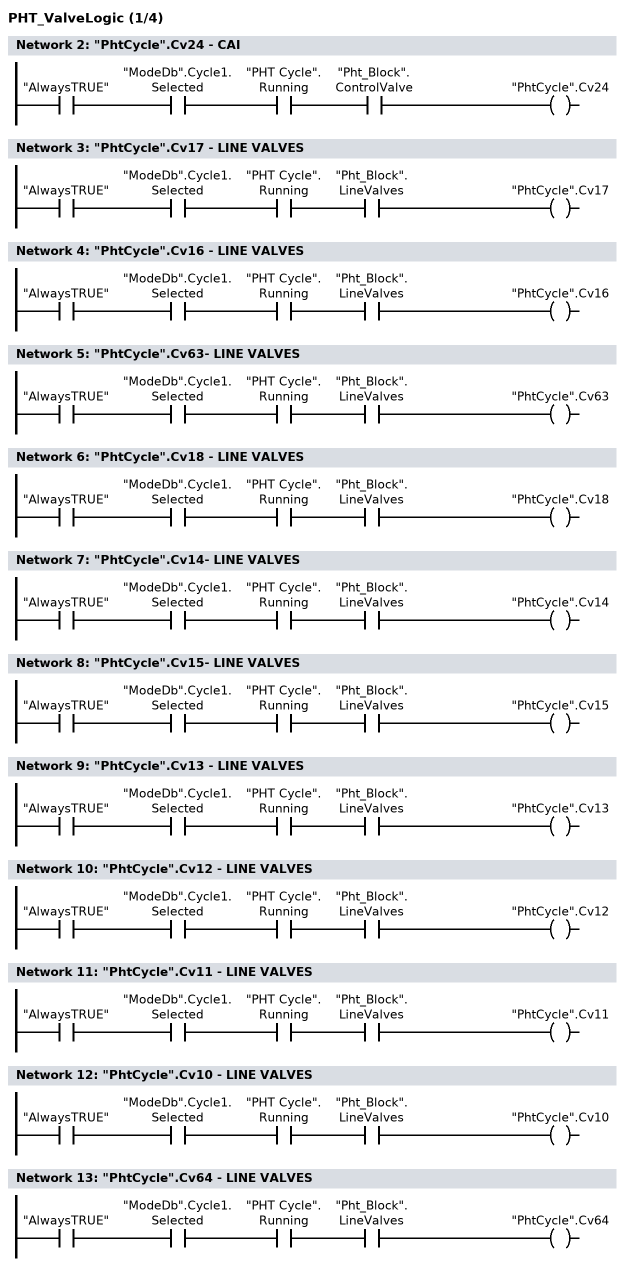
   RUNG wire#powerrail
      Contact( "AlwaysTRUE" )
      Contact( "ModeDb".Cycle1.Selected )
      Contact( "PHT Cycle".Running )
      Contact( "Pht_Block".ControlValve )
      Coil( "PhtCycle".Cv24 )
   END_RUNG
   // the same network as SCL:
   "PhtCycle".Cv24 := "AlwaysTRUE" AND "ModeDb".Cycle1.Selected AND "PHT Cycle".Running AND "Pht_Block".ControlValve;
END_REGION

REGION Network 3: "PhtCycle".Cv17 - LINE VALVES
   RUNG wire#powerrail
      Contact( "AlwaysTRUE" )
      Contact( "ModeDb".Cycle1.Selected )
      Contact( "PHT Cycle".Running )
      Contact( "Pht_Block".LineValves )
      Coil( "PhtCycle".Cv17 )
   END_RUNG
   // the same network as SCL:
   "PhtCycle".Cv17 := "AlwaysTRUE" AND "ModeDb".Cycle1.Selected AND "PHT Cycle".Running AND "Pht_Block".LineValves;
END_REGION

REGION Network 4: "PhtCycle".Cv16 - LINE VALVES
   RUNG wire#powerrail
      Contact( "AlwaysTRUE" )
      Contact( "ModeDb".Cycle1.Selected )
      Contact( "PHT Cycle".Running )
      Contact( "Pht_Block".LineValves )
      Coil( "PhtCycle".Cv16 )
   END_RUNG
   // the same network as SCL:
   "PhtCycle".Cv16 := "AlwaysTRUE" AND "ModeDb".Cycle1.Selected AND "PHT Cycle".Running AND "Pht_Block".LineValves;
END_REGION

REGION Network 5: "PhtCycle".Cv63- LINE VALVES
   RUNG wire#powerrail
      Contact( "AlwaysTRUE" )
      Contact( "ModeDb".Cycle1.Selected )
      Contact( "PHT Cycle".Running )
      Contact( "Pht_Block".LineValves )
      Coil( "PhtCycle".Cv63 )
   END_RUNG
   // the same network as SCL:
   "PhtCycle".Cv63 := "AlwaysTRUE" AND "ModeDb".Cycle1.Selected AND "PHT Cycle".Running AND "Pht_Block".LineValves;
END_REGION

REGION Network 6: "PhtCycle".Cv18 - LINE VALVES
   RUNG wire#powerrail
      Contact( "AlwaysTRUE" )
      Contact( "ModeDb".Cycle1.Selected )
      Contact( "PHT Cycle".Running )
      Contact( "Pht_Block".LineValves )
      Coil( "PhtCycle".Cv18 )
   END_RUNG
   // the same network as SCL:
   "PhtCycle".Cv18 := "AlwaysTRUE" AND "ModeDb".Cycle1.Selected AND "PHT Cycle".Running AND "Pht_Block".LineValves;
END_REGION

REGION Network 7: "PhtCycle".Cv14- LINE VALVES
   RUNG wire#powerrail
      Contact( "AlwaysTRUE" )
      Contact( "ModeDb".Cycle1.Selected )
      Contact( "PHT Cycle".Running )
      Contact( "Pht_Block".LineValves )
      Coil( "PhtCycle".Cv14 )
   END_RUNG
   // the same network as SCL:
   "PhtCycle".Cv14 := "AlwaysTRUE" AND "ModeDb".Cycle1.Selected AND "PHT Cycle".Running AND "Pht_Block".LineValves;
END_REGION

REGION Network 8: "PhtCycle".Cv15- LINE VALVES
   RUNG wire#powerrail
      Contact( "AlwaysTRUE" )
      Contact( "ModeDb".Cycle1.Selected )
      Contact( "PHT Cycle".Running )
      Contact( "Pht_Block".LineValves )
      Coil( "PhtCycle".Cv15 )
   END_RUNG
   // the same network as SCL:
   "PhtCycle".Cv15 := "AlwaysTRUE" AND "ModeDb".Cycle1.Selected AND "PHT Cycle".Running AND "Pht_Block".LineValves;
END_REGION

REGION Network 9: "PhtCycle".Cv13 - LINE VALVES
   RUNG wire#powerrail
      Contact( "AlwaysTRUE" )
      Contact( "ModeDb".Cycle1.Selected )
      Contact( "PHT Cycle".Running )
      Contact( "Pht_Block".LineValves )
      Coil( "PhtCycle".Cv13 )
   END_RUNG
   // the same network as SCL:
   "PhtCycle".Cv13 := "AlwaysTRUE" AND "ModeDb".Cycle1.Selected AND "PHT Cycle".Running AND "Pht_Block".LineValves;
END_REGION

REGION Network 10: "PhtCycle".Cv12 - LINE VALVES
   RUNG wire#powerrail
      Contact( "AlwaysTRUE" )
      Contact( "ModeDb".Cycle1.Selected )
      Contact( "PHT Cycle".Running )
      Contact( "Pht_Block".LineValves )
      Coil( "PhtCycle".Cv12 )
   END_RUNG
   // the same network as SCL:
   "PhtCycle".Cv12 := "AlwaysTRUE" AND "ModeDb".Cycle1.Selected AND "PHT Cycle".Running AND "Pht_Block".LineValves;
END_REGION

REGION Network 11: "PhtCycle".Cv11 - LINE VALVES
   RUNG wire#powerrail
      Contact( "AlwaysTRUE" )
      Contact( "ModeDb".Cycle1.Selected )
      Contact( "PHT Cycle".Running )
      Contact( "Pht_Block".LineValves )
      Coil( "PhtCycle".Cv11 )
   END_RUNG
   // the same network as SCL:
   "PhtCycle".Cv11 := "AlwaysTRUE" AND "ModeDb".Cycle1.Selected AND "PHT Cycle".Running AND "Pht_Block".LineValves;
END_REGION

REGION Network 12: "PhtCycle".Cv10 - LINE VALVES
   RUNG wire#powerrail
      Contact( "AlwaysTRUE" )
      Contact( "ModeDb".Cycle1.Selected )
      Contact( "PHT Cycle".Running )
      Contact( "Pht_Block".LineValves )
      Coil( "PhtCycle".Cv10 )
   END_RUNG
   // the same network as SCL:
   "PhtCycle".Cv10 := "AlwaysTRUE" AND "ModeDb".Cycle1.Selected AND "PHT Cycle".Running AND "Pht_Block".LineValves;
END_REGION

REGION Network 13: "PhtCycle".Cv64 - LINE VALVES
   RUNG wire#powerrail
      Contact( "AlwaysTRUE" )
      Contact( "ModeDb".Cycle1.Selected )
      Contact( "PHT Cycle".Running )
      Contact( "Pht_Block".LineValves )
      Coil( "PhtCycle".Cv64 )
   END_RUNG
   // the same network as SCL:
   "PhtCycle".Cv64 := "AlwaysTRUE" AND "ModeDb".Cycle1.Selected AND "PHT Cycle".Running AND "Pht_Block".LineValves;
END_REGION

REGION Network 14: "PhtCycle".Cv26 - LINE VALVES
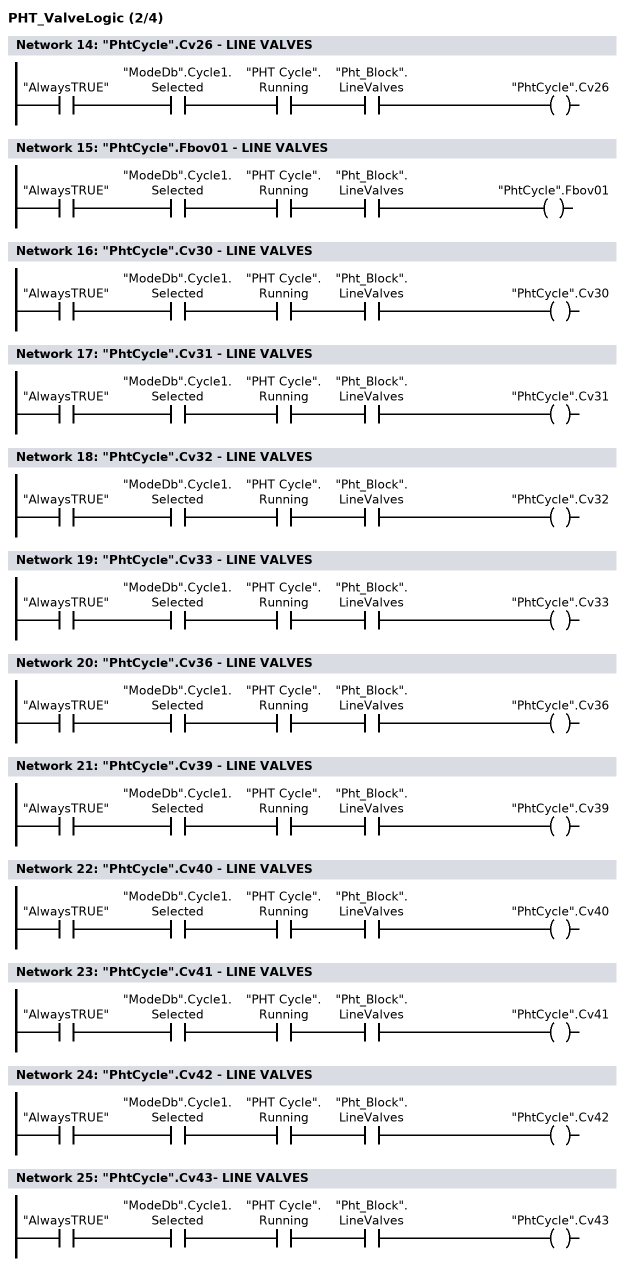
   RUNG wire#powerrail
      Contact( "AlwaysTRUE" )
      Contact( "ModeDb".Cycle1.Selected )
      Contact( "PHT Cycle".Running )
      Contact( "Pht_Block".LineValves )
      Coil( "PhtCycle".Cv26 )
   END_RUNG
   // the same network as SCL:
   "PhtCycle".Cv26 := "AlwaysTRUE" AND "ModeDb".Cycle1.Selected AND "PHT Cycle".Running AND "Pht_Block".LineValves;
END_REGION

REGION Network 15: "PhtCycle".Fbov01 - LINE VALVES
   RUNG wire#powerrail
      Contact( "AlwaysTRUE" )
      Contact( "ModeDb".Cycle1.Selected )
      Contact( "PHT Cycle".Running )
      Contact( "Pht_Block".LineValves )
      Coil( "PhtCycle".Fbov01 )
   END_RUNG
   // the same network as SCL:
   "PhtCycle".Fbov01 := "AlwaysTRUE" AND "ModeDb".Cycle1.Selected AND "PHT Cycle".Running AND "Pht_Block".LineValves;
END_REGION

REGION Network 16: "PhtCycle".Cv30 - LINE VALVES
   RUNG wire#powerrail
      Contact( "AlwaysTRUE" )
      Contact( "ModeDb".Cycle1.Selected )
      Contact( "PHT Cycle".Running )
      Contact( "Pht_Block".LineValves )
      Coil( "PhtCycle".Cv30 )
   END_RUNG
   // the same network as SCL:
   "PhtCycle".Cv30 := "AlwaysTRUE" AND "ModeDb".Cycle1.Selected AND "PHT Cycle".Running AND "Pht_Block".LineValves;
END_REGION

REGION Network 17: "PhtCycle".Cv31 - LINE VALVES
   RUNG wire#powerrail
      Contact( "AlwaysTRUE" )
      Contact( "ModeDb".Cycle1.Selected )
      Contact( "PHT Cycle".Running )
      Contact( "Pht_Block".LineValves )
      Coil( "PhtCycle".Cv31 )
   END_RUNG
   // the same network as SCL:
   "PhtCycle".Cv31 := "AlwaysTRUE" AND "ModeDb".Cycle1.Selected AND "PHT Cycle".Running AND "Pht_Block".LineValves;
END_REGION

REGION Network 18: "PhtCycle".Cv32 - LINE VALVES
   RUNG wire#powerrail
      Contact( "AlwaysTRUE" )
      Contact( "ModeDb".Cycle1.Selected )
      Contact( "PHT Cycle".Running )
      Contact( "Pht_Block".LineValves )
      Coil( "PhtCycle".Cv32 )
   END_RUNG
   // the same network as SCL:
   "PhtCycle".Cv32 := "AlwaysTRUE" AND "ModeDb".Cycle1.Selected AND "PHT Cycle".Running AND "Pht_Block".LineValves;
END_REGION

REGION Network 19: "PhtCycle".Cv33 - LINE VALVES
   RUNG wire#powerrail
      Contact( "AlwaysTRUE" )
      Contact( "ModeDb".Cycle1.Selected )
      Contact( "PHT Cycle".Running )
      Contact( "Pht_Block".LineValves )
      Coil( "PhtCycle".Cv33 )
   END_RUNG
   // the same network as SCL:
   "PhtCycle".Cv33 := "AlwaysTRUE" AND "ModeDb".Cycle1.Selected AND "PHT Cycle".Running AND "Pht_Block".LineValves;
END_REGION

REGION Network 20: "PhtCycle".Cv36 - LINE VALVES
   RUNG wire#powerrail
      Contact( "AlwaysTRUE" )
      Contact( "ModeDb".Cycle1.Selected )
      Contact( "PHT Cycle".Running )
      Contact( "Pht_Block".LineValves )
      Coil( "PhtCycle".Cv36 )
   END_RUNG
   // the same network as SCL:
   "PhtCycle".Cv36 := "AlwaysTRUE" AND "ModeDb".Cycle1.Selected AND "PHT Cycle".Running AND "Pht_Block".LineValves;
END_REGION

REGION Network 21: "PhtCycle".Cv39 - LINE VALVES
   RUNG wire#powerrail
      Contact( "AlwaysTRUE" )
      Contact( "ModeDb".Cycle1.Selected )
      Contact( "PHT Cycle".Running )
      Contact( "Pht_Block".LineValves )
      Coil( "PhtCycle".Cv39 )
   END_RUNG
   // the same network as SCL:
   "PhtCycle".Cv39 := "AlwaysTRUE" AND "ModeDb".Cycle1.Selected AND "PHT Cycle".Running AND "Pht_Block".LineValves;
END_REGION

REGION Network 22: "PhtCycle".Cv40 - LINE VALVES
   RUNG wire#powerrail
      Contact( "AlwaysTRUE" )
      Contact( "ModeDb".Cycle1.Selected )
      Contact( "PHT Cycle".Running )
      Contact( "Pht_Block".LineValves )
      Coil( "PhtCycle".Cv40 )
   END_RUNG
   // the same network as SCL:
   "PhtCycle".Cv40 := "AlwaysTRUE" AND "ModeDb".Cycle1.Selected AND "PHT Cycle".Running AND "Pht_Block".LineValves;
END_REGION

REGION Network 23: "PhtCycle".Cv41 - LINE VALVES
   RUNG wire#powerrail
      Contact( "AlwaysTRUE" )
      Contact( "ModeDb".Cycle1.Selected )
      Contact( "PHT Cycle".Running )
      Contact( "Pht_Block".LineValves )
      Coil( "PhtCycle".Cv41 )
   END_RUNG
   // the same network as SCL:
   "PhtCycle".Cv41 := "AlwaysTRUE" AND "ModeDb".Cycle1.Selected AND "PHT Cycle".Running AND "Pht_Block".LineValves;
END_REGION

REGION Network 24: "PhtCycle".Cv42 - LINE VALVES
   RUNG wire#powerrail
      Contact( "AlwaysTRUE" )
      Contact( "ModeDb".Cycle1.Selected )
      Contact( "PHT Cycle".Running )
      Contact( "Pht_Block".LineValves )
      Coil( "PhtCycle".Cv42 )
   END_RUNG
   // the same network as SCL:
   "PhtCycle".Cv42 := "AlwaysTRUE" AND "ModeDb".Cycle1.Selected AND "PHT Cycle".Running AND "Pht_Block".LineValves;
END_REGION

REGION Network 25: "PhtCycle".Cv43- LINE VALVES
   RUNG wire#powerrail
      Contact( "AlwaysTRUE" )
      Contact( "ModeDb".Cycle1.Selected )
      Contact( "PHT Cycle".Running )
      Contact( "Pht_Block".LineValves )
      Coil( "PhtCycle".Cv43 )
   END_RUNG
   // the same network as SCL:
   "PhtCycle".Cv43 := "AlwaysTRUE" AND "ModeDb".Cycle1.Selected AND "PHT Cycle".Running AND "Pht_Block".LineValves;
END_REGION

REGION Network 26: "PhtCycle".Cv44 - LINE VALVES
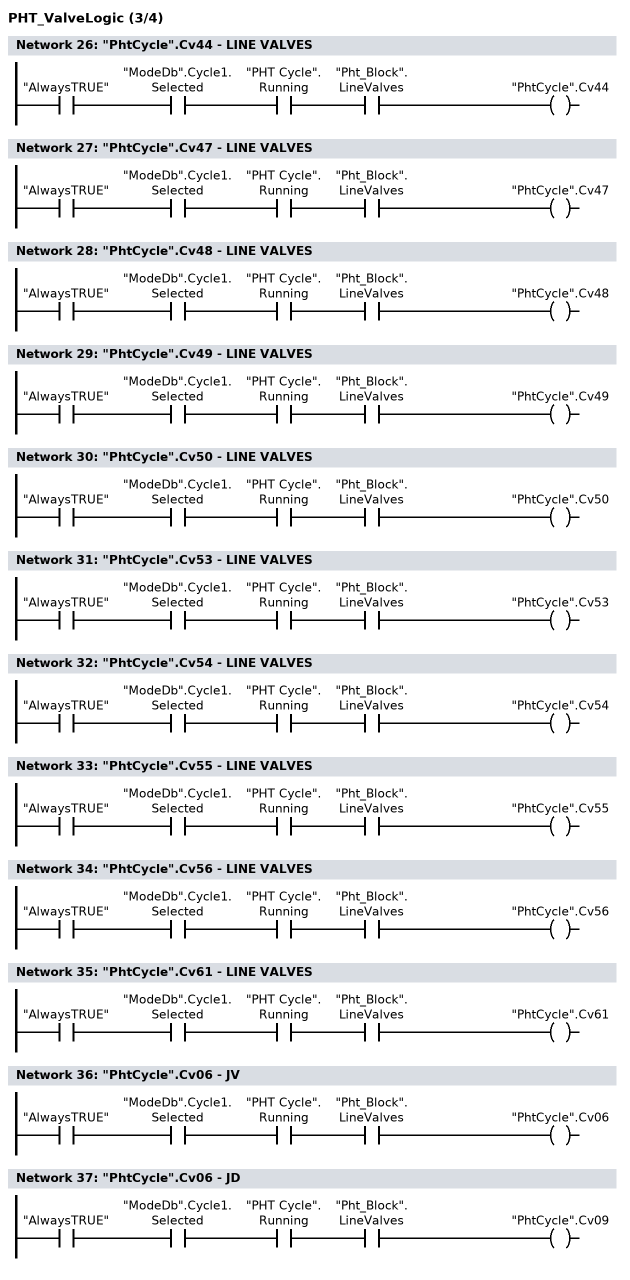
   RUNG wire#powerrail
      Contact( "AlwaysTRUE" )
      Contact( "ModeDb".Cycle1.Selected )
      Contact( "PHT Cycle".Running )
      Contact( "Pht_Block".LineValves )
      Coil( "PhtCycle".Cv44 )
   END_RUNG
   // the same network as SCL:
   "PhtCycle".Cv44 := "AlwaysTRUE" AND "ModeDb".Cycle1.Selected AND "PHT Cycle".Running AND "Pht_Block".LineValves;
END_REGION

REGION Network 27: "PhtCycle".Cv47 - LINE VALVES
   RUNG wire#powerrail
      Contact( "AlwaysTRUE" )
      Contact( "ModeDb".Cycle1.Selected )
      Contact( "PHT Cycle".Running )
      Contact( "Pht_Block".LineValves )
      Coil( "PhtCycle".Cv47 )
   END_RUNG
   // the same network as SCL:
   "PhtCycle".Cv47 := "AlwaysTRUE" AND "ModeDb".Cycle1.Selected AND "PHT Cycle".Running AND "Pht_Block".LineValves;
END_REGION

REGION Network 28: "PhtCycle".Cv48 - LINE VALVES
   RUNG wire#powerrail
      Contact( "AlwaysTRUE" )
      Contact( "ModeDb".Cycle1.Selected )
      Contact( "PHT Cycle".Running )
      Contact( "Pht_Block".LineValves )
      Coil( "PhtCycle".Cv48 )
   END_RUNG
   // the same network as SCL:
   "PhtCycle".Cv48 := "AlwaysTRUE" AND "ModeDb".Cycle1.Selected AND "PHT Cycle".Running AND "Pht_Block".LineValves;
END_REGION

REGION Network 29: "PhtCycle".Cv49 - LINE VALVES
   RUNG wire#powerrail
      Contact( "AlwaysTRUE" )
      Contact( "ModeDb".Cycle1.Selected )
      Contact( "PHT Cycle".Running )
      Contact( "Pht_Block".LineValves )
      Coil( "PhtCycle".Cv49 )
   END_RUNG
   // the same network as SCL:
   "PhtCycle".Cv49 := "AlwaysTRUE" AND "ModeDb".Cycle1.Selected AND "PHT Cycle".Running AND "Pht_Block".LineValves;
END_REGION

REGION Network 30: "PhtCycle".Cv50 - LINE VALVES
   RUNG wire#powerrail
      Contact( "AlwaysTRUE" )
      Contact( "ModeDb".Cycle1.Selected )
      Contact( "PHT Cycle".Running )
      Contact( "Pht_Block".LineValves )
      Coil( "PhtCycle".Cv50 )
   END_RUNG
   // the same network as SCL:
   "PhtCycle".Cv50 := "AlwaysTRUE" AND "ModeDb".Cycle1.Selected AND "PHT Cycle".Running AND "Pht_Block".LineValves;
END_REGION

REGION Network 31: "PhtCycle".Cv53 - LINE VALVES
   RUNG wire#powerrail
      Contact( "AlwaysTRUE" )
      Contact( "ModeDb".Cycle1.Selected )
      Contact( "PHT Cycle".Running )
      Contact( "Pht_Block".LineValves )
      Coil( "PhtCycle".Cv53 )
   END_RUNG
   // the same network as SCL:
   "PhtCycle".Cv53 := "AlwaysTRUE" AND "ModeDb".Cycle1.Selected AND "PHT Cycle".Running AND "Pht_Block".LineValves;
END_REGION

REGION Network 32: "PhtCycle".Cv54 - LINE VALVES
   RUNG wire#powerrail
      Contact( "AlwaysTRUE" )
      Contact( "ModeDb".Cycle1.Selected )
      Contact( "PHT Cycle".Running )
      Contact( "Pht_Block".LineValves )
      Coil( "PhtCycle".Cv54 )
   END_RUNG
   // the same network as SCL:
   "PhtCycle".Cv54 := "AlwaysTRUE" AND "ModeDb".Cycle1.Selected AND "PHT Cycle".Running AND "Pht_Block".LineValves;
END_REGION

REGION Network 33: "PhtCycle".Cv55 - LINE VALVES
   RUNG wire#powerrail
      Contact( "AlwaysTRUE" )
      Contact( "ModeDb".Cycle1.Selected )
      Contact( "PHT Cycle".Running )
      Contact( "Pht_Block".LineValves )
      Coil( "PhtCycle".Cv55 )
   END_RUNG
   // the same network as SCL:
   "PhtCycle".Cv55 := "AlwaysTRUE" AND "ModeDb".Cycle1.Selected AND "PHT Cycle".Running AND "Pht_Block".LineValves;
END_REGION

REGION Network 34: "PhtCycle".Cv56 - LINE VALVES
   RUNG wire#powerrail
      Contact( "AlwaysTRUE" )
      Contact( "ModeDb".Cycle1.Selected )
      Contact( "PHT Cycle".Running )
      Contact( "Pht_Block".LineValves )
      Coil( "PhtCycle".Cv56 )
   END_RUNG
   // the same network as SCL:
   "PhtCycle".Cv56 := "AlwaysTRUE" AND "ModeDb".Cycle1.Selected AND "PHT Cycle".Running AND "Pht_Block".LineValves;
END_REGION

REGION Network 35: "PhtCycle".Cv61 - LINE VALVES
   RUNG wire#powerrail
      Contact( "AlwaysTRUE" )
      Contact( "ModeDb".Cycle1.Selected )
      Contact( "PHT Cycle".Running )
      Contact( "Pht_Block".LineValves )
      Coil( "PhtCycle".Cv61 )
   END_RUNG
   // the same network as SCL:
   "PhtCycle".Cv61 := "AlwaysTRUE" AND "ModeDb".Cycle1.Selected AND "PHT Cycle".Running AND "Pht_Block".LineValves;
END_REGION

REGION Network 36: "PhtCycle".Cv06 - JV
   RUNG wire#powerrail
      Contact( "AlwaysTRUE" )
      Contact( "ModeDb".Cycle1.Selected )
      Contact( "PHT Cycle".Running )
      Contact( "Pht_Block".LineValves )
      Coil( "PhtCycle".Cv06 )
   END_RUNG
   // the same network as SCL:
   "PhtCycle".Cv06 := "AlwaysTRUE" AND "ModeDb".Cycle1.Selected AND "PHT Cycle".Running AND "Pht_Block".LineValves;
END_REGION

REGION Network 37: "PhtCycle".Cv06 - JD
   RUNG wire#powerrail
      Contact( "AlwaysTRUE" )
      Contact( "ModeDb".Cycle1.Selected )
      Contact( "PHT Cycle".Running )
      Contact( "Pht_Block".LineValves )
      Coil( "PhtCycle".Cv09 )
   END_RUNG
   // the same network as SCL:
   "PhtCycle".Cv09 := "AlwaysTRUE" AND "ModeDb".Cycle1.Selected AND "PHT Cycle".Running AND "Pht_Block".LineValves;
END_REGION

REGION Network 38: ________________________________RELEASE VALVE________________________________
END_REGION

REGION Network 39: "PhtCycle".Cv25 - RELEASE VALVE
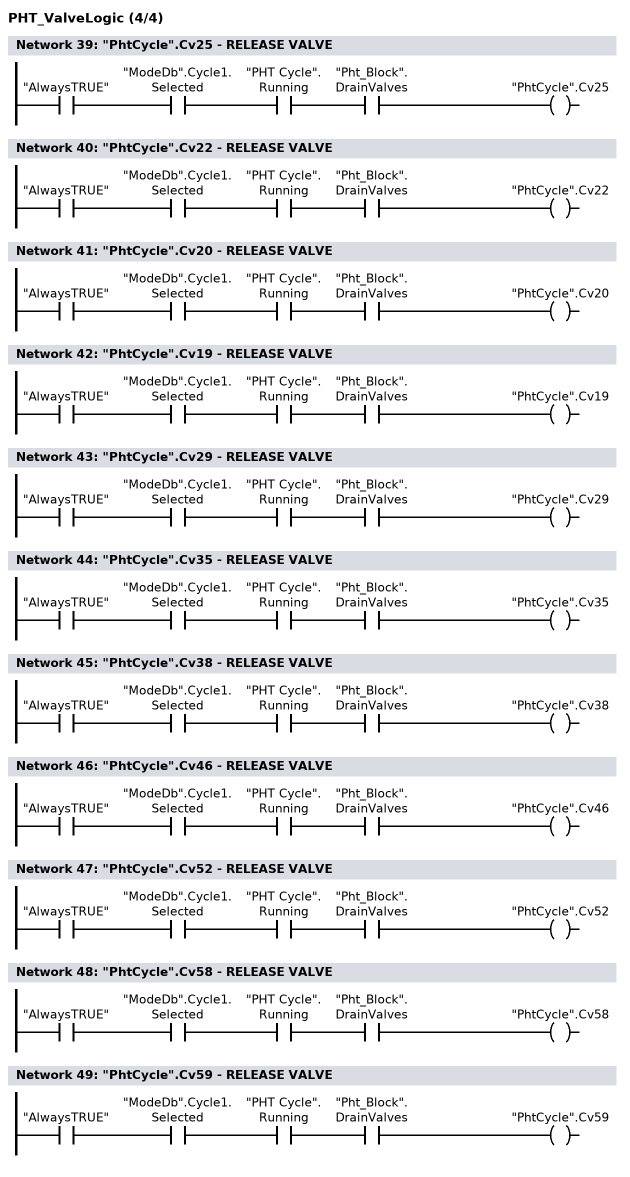
   RUNG wire#powerrail
      Contact( "AlwaysTRUE" )
      Contact( "ModeDb".Cycle1.Selected )
      Contact( "PHT Cycle".Running )
      Contact( "Pht_Block".DrainValves )
      Coil( "PhtCycle".Cv25 )
   END_RUNG
   // the same network as SCL:
   "PhtCycle".Cv25 := "AlwaysTRUE" AND "ModeDb".Cycle1.Selected AND "PHT Cycle".Running AND "Pht_Block".DrainValves;
END_REGION

REGION Network 40: "PhtCycle".Cv22 - RELEASE VALVE
   RUNG wire#powerrail
      Contact( "AlwaysTRUE" )
      Contact( "ModeDb".Cycle1.Selected )
      Contact( "PHT Cycle".Running )
      Contact( "Pht_Block".DrainValves )
      Coil( "PhtCycle".Cv22 )
   END_RUNG
   // the same network as SCL:
   "PhtCycle".Cv22 := "AlwaysTRUE" AND "ModeDb".Cycle1.Selected AND "PHT Cycle".Running AND "Pht_Block".DrainValves;
END_REGION

REGION Network 41: "PhtCycle".Cv20 - RELEASE VALVE
   RUNG wire#powerrail
      Contact( "AlwaysTRUE" )
      Contact( "ModeDb".Cycle1.Selected )
      Contact( "PHT Cycle".Running )
      Contact( "Pht_Block".DrainValves )
      Coil( "PhtCycle".Cv20 )
   END_RUNG
   // the same network as SCL:
   "PhtCycle".Cv20 := "AlwaysTRUE" AND "ModeDb".Cycle1.Selected AND "PHT Cycle".Running AND "Pht_Block".DrainValves;
END_REGION

REGION Network 42: "PhtCycle".Cv19 - RELEASE VALVE
   RUNG wire#powerrail
      Contact( "AlwaysTRUE" )
      Contact( "ModeDb".Cycle1.Selected )
      Contact( "PHT Cycle".Running )
      Contact( "Pht_Block".DrainValves )
      Coil( "PhtCycle".Cv19 )
   END_RUNG
   // the same network as SCL:
   "PhtCycle".Cv19 := "AlwaysTRUE" AND "ModeDb".Cycle1.Selected AND "PHT Cycle".Running AND "Pht_Block".DrainValves;
END_REGION

REGION Network 43: "PhtCycle".Cv29 - RELEASE VALVE
   RUNG wire#powerrail
      Contact( "AlwaysTRUE" )
      Contact( "ModeDb".Cycle1.Selected )
      Contact( "PHT Cycle".Running )
      Contact( "Pht_Block".DrainValves )
      Coil( "PhtCycle".Cv29 )
   END_RUNG
   // the same network as SCL:
   "PhtCycle".Cv29 := "AlwaysTRUE" AND "ModeDb".Cycle1.Selected AND "PHT Cycle".Running AND "Pht_Block".DrainValves;
END_REGION

REGION Network 44: "PhtCycle".Cv35 - RELEASE VALVE
   RUNG wire#powerrail
      Contact( "AlwaysTRUE" )
      Contact( "ModeDb".Cycle1.Selected )
      Contact( "PHT Cycle".Running )
      Contact( "Pht_Block".DrainValves )
      Coil( "PhtCycle".Cv35 )
   END_RUNG
   // the same network as SCL:
   "PhtCycle".Cv35 := "AlwaysTRUE" AND "ModeDb".Cycle1.Selected AND "PHT Cycle".Running AND "Pht_Block".DrainValves;
END_REGION

REGION Network 45: "PhtCycle".Cv38 - RELEASE VALVE
   RUNG wire#powerrail
      Contact( "AlwaysTRUE" )
      Contact( "ModeDb".Cycle1.Selected )
      Contact( "PHT Cycle".Running )
      Contact( "Pht_Block".DrainValves )
      Coil( "PhtCycle".Cv38 )
   END_RUNG
   // the same network as SCL:
   "PhtCycle".Cv38 := "AlwaysTRUE" AND "ModeDb".Cycle1.Selected AND "PHT Cycle".Running AND "Pht_Block".DrainValves;
END_REGION

REGION Network 46: "PhtCycle".Cv46 - RELEASE VALVE
   RUNG wire#powerrail
      Contact( "AlwaysTRUE" )
      Contact( "ModeDb".Cycle1.Selected )
      Contact( "PHT Cycle".Running )
      Contact( "Pht_Block".DrainValves )
      Coil( "PhtCycle".Cv46 )
   END_RUNG
   // the same network as SCL:
   "PhtCycle".Cv46 := "AlwaysTRUE" AND "ModeDb".Cycle1.Selected AND "PHT Cycle".Running AND "Pht_Block".DrainValves;
END_REGION

REGION Network 47: "PhtCycle".Cv52 - RELEASE VALVE
   RUNG wire#powerrail
      Contact( "AlwaysTRUE" )
      Contact( "ModeDb".Cycle1.Selected )
      Contact( "PHT Cycle".Running )
      Contact( "Pht_Block".DrainValves )
      Coil( "PhtCycle".Cv52 )
   END_RUNG
   // the same network as SCL:
   "PhtCycle".Cv52 := "AlwaysTRUE" AND "ModeDb".Cycle1.Selected AND "PHT Cycle".Running AND "Pht_Block".DrainValves;
END_REGION

REGION Network 48: "PhtCycle".Cv58 - RELEASE VALVE
   RUNG wire#powerrail
      Contact( "AlwaysTRUE" )
      Contact( "ModeDb".Cycle1.Selected )
      Contact( "PHT Cycle".Running )
      Contact( "Pht_Block".DrainValves )
      Coil( "PhtCycle".Cv58 )
   END_RUNG
   // the same network as SCL:
   "PhtCycle".Cv58 := "AlwaysTRUE" AND "ModeDb".Cycle1.Selected AND "PHT Cycle".Running AND "Pht_Block".DrainValves;
END_REGION

REGION Network 49: "PhtCycle".Cv59 - RELEASE VALVE
   RUNG wire#powerrail
      Contact( "AlwaysTRUE" )
      Contact( "ModeDb".Cycle1.Selected )
      Contact( "PHT Cycle".Running )
      Contact( "Pht_Block".DrainValves )
      Coil( "PhtCycle".Cv59 )
   END_RUNG
   // the same network as SCL:
   "PhtCycle".Cv59 := "AlwaysTRUE" AND "ModeDb".Cycle1.Selected AND "PHT Cycle".Running AND "Pht_Block".DrainValves;
END_REGION
END_FUNCTION

FUNCTION "LineAnimationFC" : Void   // FC311, LAD
{ S7_Optimized_Access := 'TRUE' }
// stored: AutoNumber false, SetENOAutomatically false
BEGIN

REGION Network 1: "LineAnimationDb"
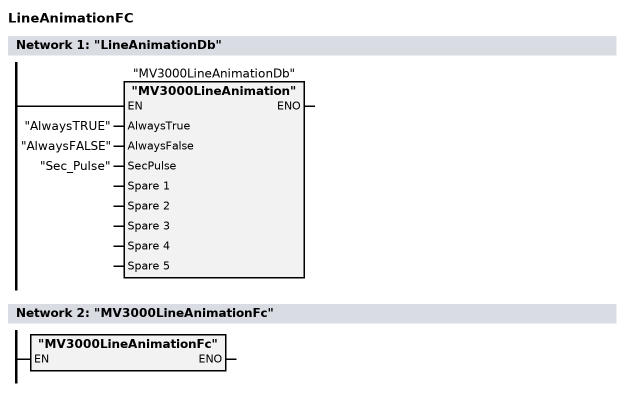
   RUNG wire#powerrail
      "MV3000LineAnimationDb"(AlwaysTrue := "AlwaysTRUE", AlwaysFalse := "AlwaysFALSE", SecPulse := "Sec_Pulse", "Spare 1" :=, "Spare 2" :=, "Spare 3" :=, "Spare 4" :=, "Spare 5" :=)
   END_RUNG
   // the same network as SCL:
   "MV3000LineAnimationDb"(AlwaysTrue := "AlwaysTRUE", AlwaysFalse := "AlwaysFALSE", SecPulse := "Sec_Pulse");   // "MV3000LineAnimation"
END_REGION

REGION Network 2: "MV3000LineAnimationFc"
   RUNG wire#powerrail
      "MV3000LineAnimationFc"()
   END_RUNG
   // the same network as SCL:
   "MV3000LineAnimationFc"();
END_REGION
END_FUNCTION

FUNCTION_BLOCK "MV3000LineAnimation"   // FB801, LAD
{ S7_Optimized_Access := 'FALSE' }
// stored: AutoNumber false, SetENOAutomatically false
   VAR_INPUT
      AlwaysTrue : Bool;
      AlwaysFalse : Bool;
      SecPulse : Bool;
      "Spare 1" : Bool;
      "Spare 2" : Bool;
      "Spare 3" : Bool;
      "Spare 4" : Bool;
      "Spare 5" : Bool;
   END_VAR
   VAR
      "Node 1" : "LineAnimationFb";
      "Node 2" : "LineAnimationFb";
      "Node 3" : "LineAnimationFb";
      "Node 4" : "LineAnimationFb";
      "Node 5" : "LineAnimationFb";
      "Node 6" : "LineAnimationFb";
      "Node 7" { S7_SetPoint := 'True'} : "LineAnimationFb";
      "Node 8" { S7_SetPoint := 'True'} : "LineAnimationFb";
      "Node 9" { S7_SetPoint := 'True'} : "LineAnimationFb";
      "Node 10" { S7_SetPoint := 'True'} : "LineAnimationFb";
      "Node 11" { S7_SetPoint := 'True'} : "LineAnimationFb";
      "Node 12" { S7_SetPoint := 'True'} : "LineAnimationFb";
      "Node 13" { S7_SetPoint := 'True'} : "LineAnimationFb";
      "Node 14" { S7_SetPoint := 'True'} : "LineAnimationFb";
      "Node 15" { S7_SetPoint := 'True'} : "LineAnimationFb";
      "Node 16" { S7_SetPoint := 'True'} : "LineAnimationFb";
      "Node 17" { S7_SetPoint := 'True'} : "LineAnimationFb";
      "Node 18" { S7_SetPoint := 'True'} : "LineAnimationFb";
      "Node 19" { S7_SetPoint := 'True'} : "LineAnimationFb";
      "Node 20" { S7_SetPoint := 'True'} : "LineAnimationFb";
      "Node 21" { S7_SetPoint := 'True'} : "LineAnimationFb";
      "Node 22" { S7_SetPoint := 'True'} : "LineAnimationFb";
      "Node 23" { S7_SetPoint := 'True'} : "LineAnimationFb";
      "Node 24" { S7_SetPoint := 'True'} : "LineAnimationFb";
      "Node 25" { S7_SetPoint := 'True'} : "LineAnimationFb";
      "Node 26" { S7_SetPoint := 'True'} : "LineAnimationFb";
      "Node 27" { S7_SetPoint := 'True'} : "LineAnimationFb";
      "Node 28" { S7_SetPoint := 'True'} : "LineAnimationFb";
      "Node 29" { S7_SetPoint := 'True'} : "LineAnimationFb";
      "Node 30" { S7_SetPoint := 'True'} : "LineAnimationFb";
      Node31 { S7_SetPoint := 'True'} : "LineAnimationFb";
      Node32 { S7_SetPoint := 'True'} : "LineAnimationFb";
      Node33 { S7_SetPoint := 'True'} : "LineAnimationFb";
      Node34 { S7_SetPoint := 'True'} : "LineAnimationFb";
   END_VAR
BEGIN

REGION Network 1: Cv01,Cv02, Cv10
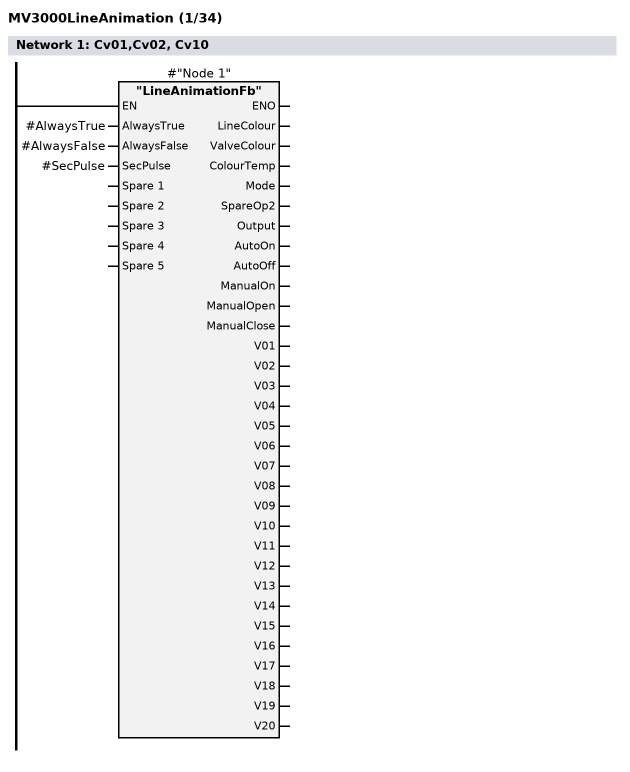
   RUNG wire#powerrail
      #"Node 1"(AlwaysTrue := #AlwaysTrue, AlwaysFalse := #AlwaysFalse, SecPulse := #SecPulse, "Spare 1" :=, "Spare 2" :=, "Spare 3" :=, "Spare 4" :=, "Spare 5" :=, LineColour =>, ValveColour =>, ColourTemp =>, Mode =>, SpareOp2 =>, Output =>, AutoOn =>, AutoOff =>, ManualOn =>, ManualOpen =>, ManualClose =>, V01 =>, V02 =>, V03 =>, V04 =>, V05 =>, V06 =>, V07 =>, V08 =>, V09 =>, V10 =>, V11 =>, V12 =>, V13 =>, V14 =>, V15 =>, V16 =>, V17 =>, V18 =>, V19 =>, V20 =>)
   END_RUNG
   // the same network as SCL:
   #"Node 1"(AlwaysTrue := #AlwaysTrue, AlwaysFalse := #AlwaysFalse, SecPulse := #SecPulse);   // "LineAnimationFb"
END_REGION

REGION Network 2: Cv03,Cv04,Cv05,Cv06
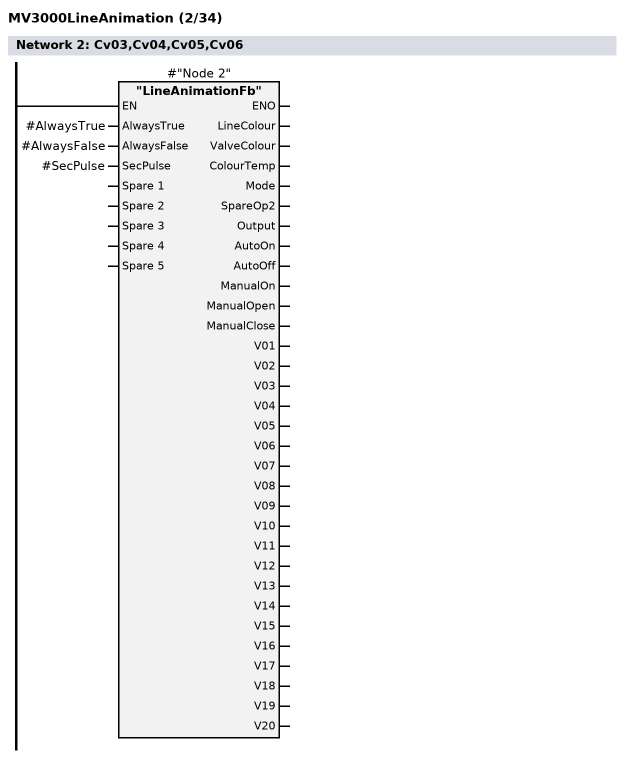
   RUNG wire#powerrail
      #"Node 2"(AlwaysTrue := #AlwaysTrue, AlwaysFalse := #AlwaysFalse, SecPulse := #SecPulse, "Spare 1" :=, "Spare 2" :=, "Spare 3" :=, "Spare 4" :=, "Spare 5" :=, LineColour =>, ValveColour =>, ColourTemp =>, Mode =>, SpareOp2 =>, Output =>, AutoOn =>, AutoOff =>, ManualOn =>, ManualOpen =>, ManualClose =>, V01 =>, V02 =>, V03 =>, V04 =>, V05 =>, V06 =>, V07 =>, V08 =>, V09 =>, V10 =>, V11 =>, V12 =>, V13 =>, V14 =>, V15 =>, V16 =>, V17 =>, V18 =>, V19 =>, V20 =>)
   END_RUNG
   // the same network as SCL:
   #"Node 2"(AlwaysTrue := #AlwaysTrue, AlwaysFalse := #AlwaysFalse, SecPulse := #SecPulse);   // "LineAnimationFb"
END_REGION

REGION Network 3: Cv07,Cv08, Cv09
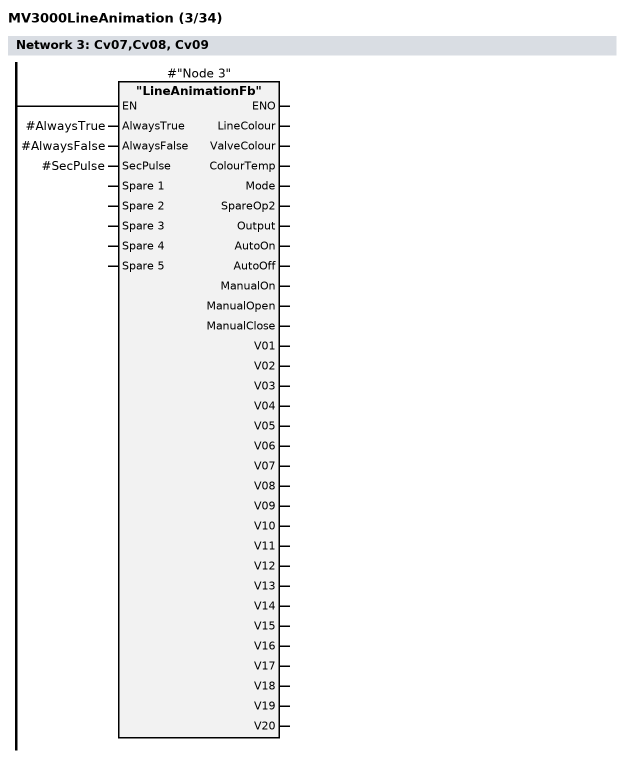
   RUNG wire#powerrail
      #"Node 3"(AlwaysTrue := #AlwaysTrue, AlwaysFalse := #AlwaysFalse, SecPulse := #SecPulse, "Spare 1" :=, "Spare 2" :=, "Spare 3" :=, "Spare 4" :=, "Spare 5" :=, LineColour =>, ValveColour =>, ColourTemp =>, Mode =>, SpareOp2 =>, Output =>, AutoOn =>, AutoOff =>, ManualOn =>, ManualOpen =>, ManualClose =>, V01 =>, V02 =>, V03 =>, V04 =>, V05 =>, V06 =>, V07 =>, V08 =>, V09 =>, V10 =>, V11 =>, V12 =>, V13 =>, V14 =>, V15 =>, V16 =>, V17 =>, V18 =>, V19 =>, V20 =>)
   END_RUNG
   // the same network as SCL:
   #"Node 3"(AlwaysTrue := #AlwaysTrue, AlwaysFalse := #AlwaysFalse, SecPulse := #SecPulse);   // "LineAnimationFb"
END_REGION

REGION Network 4: Cv16,Cv17,Cv22,Cv23,Cv24,Cv25
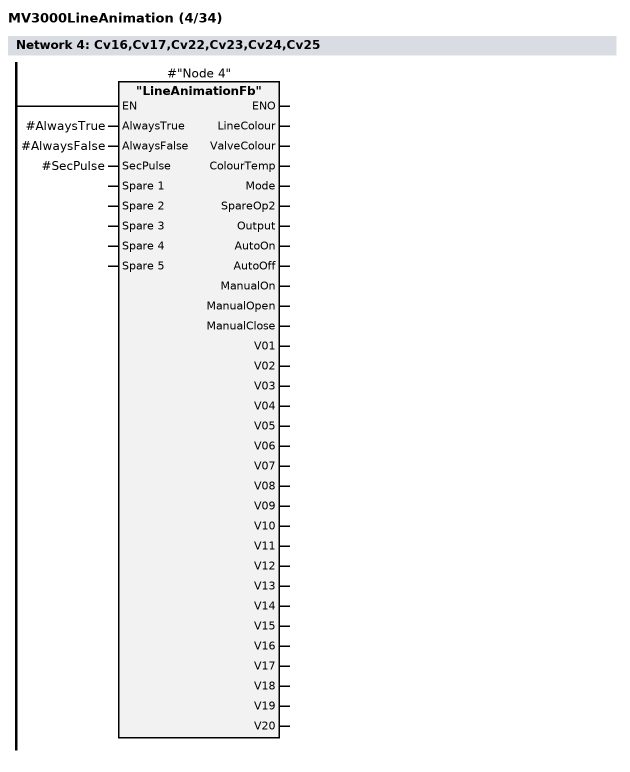
   RUNG wire#powerrail
      #"Node 4"(AlwaysTrue := #AlwaysTrue, AlwaysFalse := #AlwaysFalse, SecPulse := #SecPulse, "Spare 1" :=, "Spare 2" :=, "Spare 3" :=, "Spare 4" :=, "Spare 5" :=, LineColour =>, ValveColour =>, ColourTemp =>, Mode =>, SpareOp2 =>, Output =>, AutoOn =>, AutoOff =>, ManualOn =>, ManualOpen =>, ManualClose =>, V01 =>, V02 =>, V03 =>, V04 =>, V05 =>, V06 =>, V07 =>, V08 =>, V09 =>, V10 =>, V11 =>, V12 =>, V13 =>, V14 =>, V15 =>, V16 =>, V17 =>, V18 =>, V19 =>, V20 =>)
   END_RUNG
   // the same network as SCL:
   #"Node 4"(AlwaysTrue := #AlwaysTrue, AlwaysFalse := #AlwaysFalse, SecPulse := #SecPulse);   // "LineAnimationFb"
END_REGION

REGION Network 5: Cv22,Cv25
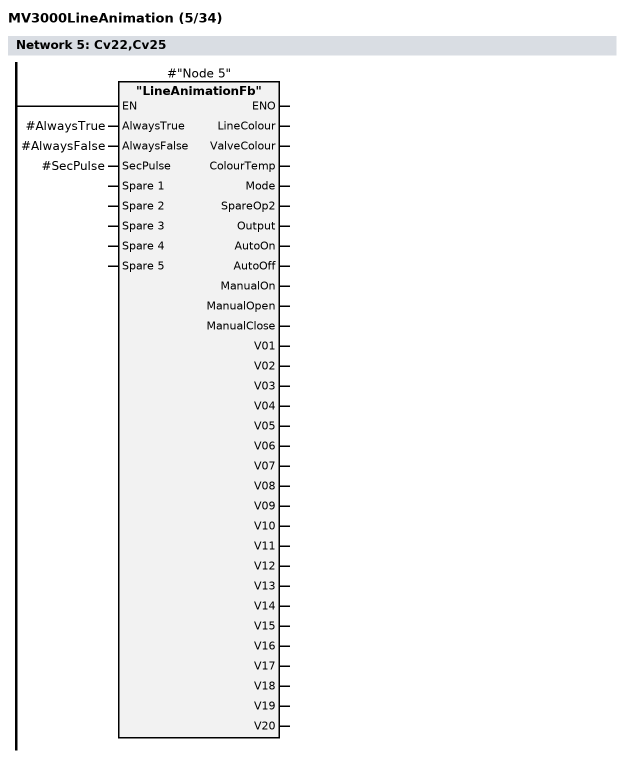
   RUNG wire#powerrail
      #"Node 5"(AlwaysTrue := #AlwaysTrue, AlwaysFalse := #AlwaysFalse, SecPulse := #SecPulse, "Spare 1" :=, "Spare 2" :=, "Spare 3" :=, "Spare 4" :=, "Spare 5" :=, LineColour =>, ValveColour =>, ColourTemp =>, Mode =>, SpareOp2 =>, Output =>, AutoOn =>, AutoOff =>, ManualOn =>, ManualOpen =>, ManualClose =>, V01 =>, V02 =>, V03 =>, V04 =>, V05 =>, V06 =>, V07 =>, V08 =>, V09 =>, V10 =>, V11 =>, V12 =>, V13 =>, V14 =>, V15 =>, V16 =>, V17 =>, V18 =>, V19 =>, V20 =>)
   END_RUNG
   // the same network as SCL:
   #"Node 5"(AlwaysTrue := #AlwaysTrue, AlwaysFalse := #AlwaysFalse, SecPulse := #SecPulse);   // "LineAnimationFb"
END_REGION

REGION Network 6: Cv18,Cv19,Cv20,Cv21
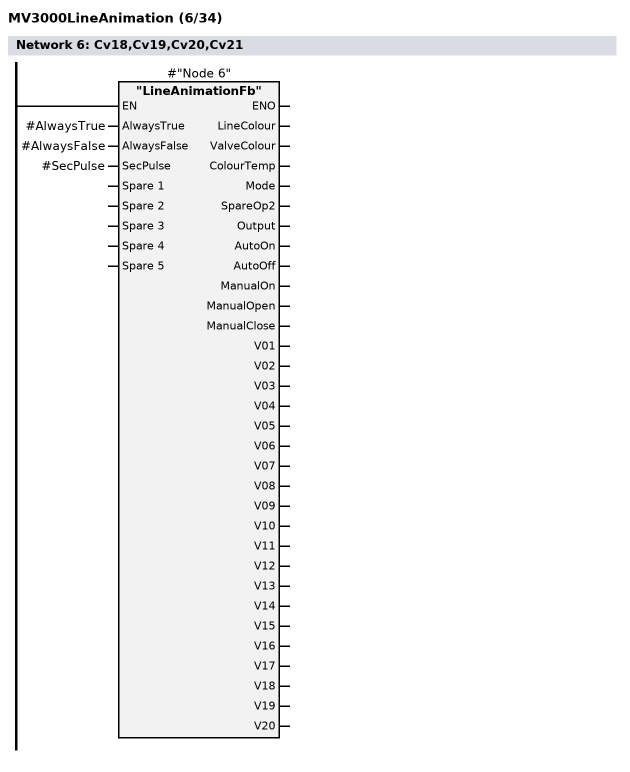
   RUNG wire#powerrail
      #"Node 6"(AlwaysTrue := #AlwaysTrue, AlwaysFalse := #AlwaysFalse, SecPulse := #SecPulse, "Spare 1" :=, "Spare 2" :=, "Spare 3" :=, "Spare 4" :=, "Spare 5" :=, LineColour =>, ValveColour =>, ColourTemp =>, Mode =>, SpareOp2 =>, Output =>, AutoOn =>, AutoOff =>, ManualOn =>, ManualOpen =>, ManualClose =>, V01 =>, V02 =>, V03 =>, V04 =>, V05 =>, V06 =>, V07 =>, V08 =>, V09 =>, V10 =>, V11 =>, V12 =>, V13 =>, V14 =>, V15 =>, V16 =>, V17 =>, V18 =>, V19 =>, V20 =>)
   END_RUNG
   // the same network as SCL:
   #"Node 6"(AlwaysTrue := #AlwaysTrue, AlwaysFalse := #AlwaysFalse, SecPulse := #SecPulse);   // "LineAnimationFb"
END_REGION

REGION Network 7: Cv19,Cv20
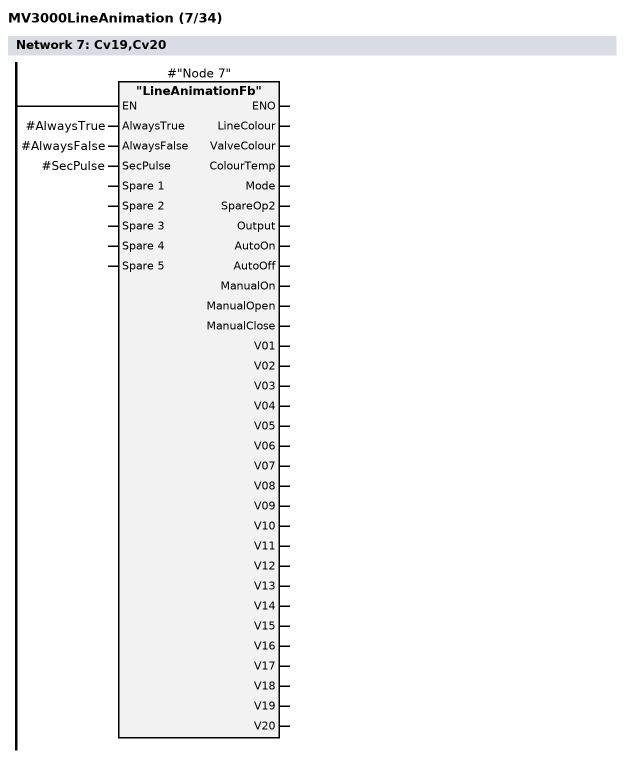
   RUNG wire#powerrail
      #"Node 7"(AlwaysTrue := #AlwaysTrue, AlwaysFalse := #AlwaysFalse, SecPulse := #SecPulse, "Spare 1" :=, "Spare 2" :=, "Spare 3" :=, "Spare 4" :=, "Spare 5" :=, LineColour =>, ValveColour =>, ColourTemp =>, Mode =>, SpareOp2 =>, Output =>, AutoOn =>, AutoOff =>, ManualOn =>, ManualOpen =>, ManualClose =>, V01 =>, V02 =>, V03 =>, V04 =>, V05 =>, V06 =>, V07 =>, V08 =>, V09 =>, V10 =>, V11 =>, V12 =>, V13 =>, V14 =>, V15 =>, V16 =>, V17 =>, V18 =>, V19 =>, V20 =>)
   END_RUNG
   // the same network as SCL:
   #"Node 7"(AlwaysTrue := #AlwaysTrue, AlwaysFalse := #AlwaysFalse, SecPulse := #SecPulse);   // "LineAnimationFb"
END_REGION

REGION Network 8: Cv16,Cv63, Cv15
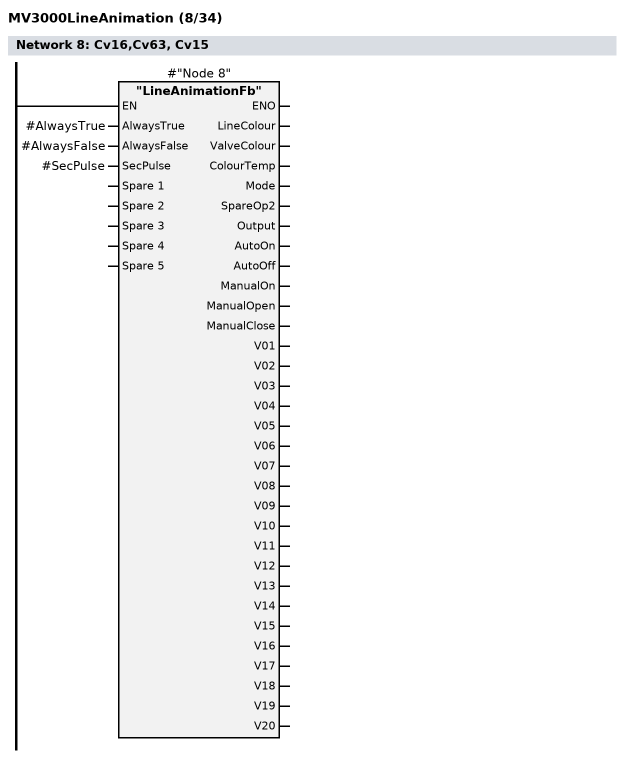
   RUNG wire#powerrail
      #"Node 8"(AlwaysTrue := #AlwaysTrue, AlwaysFalse := #AlwaysFalse, SecPulse := #SecPulse, "Spare 1" :=, "Spare 2" :=, "Spare 3" :=, "Spare 4" :=, "Spare 5" :=, LineColour =>, ValveColour =>, ColourTemp =>, Mode =>, SpareOp2 =>, Output =>, AutoOn =>, AutoOff =>, ManualOn =>, ManualOpen =>, ManualClose =>, V01 =>, V02 =>, V03 =>, V04 =>, V05 =>, V06 =>, V07 =>, V08 =>, V09 =>, V10 =>, V11 =>, V12 =>, V13 =>, V14 =>, V15 =>, V16 =>, V17 =>, V18 =>, V19 =>, V20 =>)
   END_RUNG
   // the same network as SCL:
   #"Node 8"(AlwaysTrue := #AlwaysTrue, AlwaysFalse := #AlwaysFalse, SecPulse := #SecPulse);   // "LineAnimationFb"
END_REGION

REGION Network 9: Cv10,Cv11,Cv12,Cv13,Cv14,Cv15
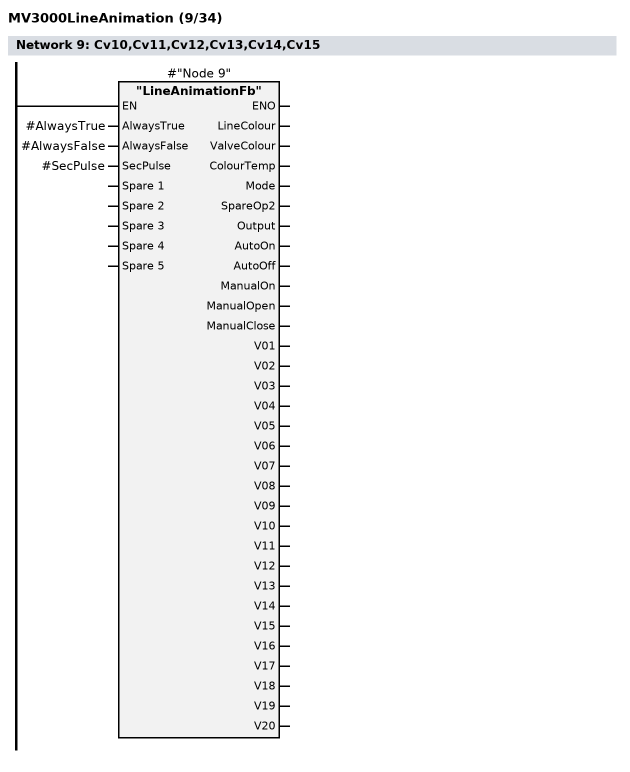
   RUNG wire#powerrail
      #"Node 9"(AlwaysTrue := #AlwaysTrue, AlwaysFalse := #AlwaysFalse, SecPulse := #SecPulse, "Spare 1" :=, "Spare 2" :=, "Spare 3" :=, "Spare 4" :=, "Spare 5" :=, LineColour =>, ValveColour =>, ColourTemp =>, Mode =>, SpareOp2 =>, Output =>, AutoOn =>, AutoOff =>, ManualOn =>, ManualOpen =>, ManualClose =>, V01 =>, V02 =>, V03 =>, V04 =>, V05 =>, V06 =>, V07 =>, V08 =>, V09 =>, V10 =>, V11 =>, V12 =>, V13 =>, V14 =>, V15 =>, V16 =>, V17 =>, V18 =>, V19 =>, V20 =>)
   END_RUNG
   // the same network as SCL:
   #"Node 9"(AlwaysTrue := #AlwaysTrue, AlwaysFalse := #AlwaysFalse, SecPulse := #SecPulse);   // "LineAnimationFb"
END_REGION

REGION Network 10: Cv11,Cv39
